    movel([0.104510, -1.367756, -2.579671, -0.764962, 1.570796, 1.675306],accel_mss,speed_ms,0,blend_radius_m)
    movel([0.104276, -1.367419, -2.579903, -0.765067, 1.570796, 1.675072],accel_mss,speed_ms,0,blend_radius_m)
    movel([0.103915, -1.367320, -2.579970, -0.765098, 1.570796, 1.674711],accel_mss,speed_ms,0,blend_radius_m)
    movel([0.103332, -1.367539, -2.579820, -0.765030, 1.570796, 1.674129],accel_mss,speed_ms,0,blend_radius_m)
    movel([0.102835, -1.367799, -2.579641, -0.764949, 1.570796, 1.673632],accel_mss,speed_ms,0,blend_radius_m)
    movel([0.102185, -1.368173, -2.579384, -0.764832, 1.570796, 1.672982],accel_mss,speed_ms,0,blend_radius_m)
    movel([0.099075, -1.369824, -2.578246, -0.764320, 1.570796, 1.669871],accel_mss,speed_ms,0,blend_radius_m)
    movel([0.095590, -1.371345, -2.577193, -0.763851, 1.570796, 1.666387],accel_mss,speed_ms,0,blend_radius_m)
    movel([0.091812, -1.372711, -2.576245, -0.763432, 1.570796, 1.662609],accel_mss,speed_ms,0,blend_radius_m)
    movel([0.087807, -1.373897, -2.575421, -0.763072, 1.570796, 1.658604],accel_mss,speed_ms,0,blend_radius_m)
    movel([0.084957, -1.374600, -2.574930, -0.762858, 1.570796, 1.655753],accel_mss,speed_ms,0,blend_radius_m)
    movel([0.082581, -1.375066, -2.574606, -0.762718, 1.570796, 1.653377],accel_mss,speed_ms,0,blend_radius_m)
    movel([0.080422, -1.375336, -2.574417, -0.762636, 1.570796, 1.651219],accel_mss,speed_ms,0,blend_radius_m)
    movel([0.078241, -1.375448, -2.574339, -0.762603, 1.570796, 1.649037],accel_mss,speed_ms,0,blend_radius_m)
    movel([0.077595, -1.375463, -2.574328, -0.762598, 1.570796, 1.648391],accel_mss,speed_ms,0,blend_radius_m)
    movel([0.077017, -1.375486, -2.574312, -0.762591, 1.570796, 1.647813],accel_mss,speed_ms,0,blend_radius_m)
    movel([0.076527, -1.375514, -2.574293, -0.762583, 1.570796, 1.647323],accel_mss,speed_ms,0,blend_radius_m)
    movel([0.076144, -1.375675, -2.574180, -0.762534, 1.570796, 1.646941],accel_mss,speed_ms,0,blend_radius_m)
    movel([0.075861, -1.375963, -2.573979, -0.762448, 1.570796, 1.646658],accel_mss,speed_ms,0,blend_radius_m)
    movel([0.075599, -1.376321, -2.573728, -0.762340, 1.570796, 1.646396],accel_mss,speed_ms,0,blend_radius_m)
    movel([0.075421, -1.376678, -2.573478, -0.762233, 1.570796, 1.646217],accel_mss,speed_ms,0,blend_radius_m)
    movel([0.075249, -1.377242, -2.573082, -0.762064, 1.570796, 1.646045],accel_mss,speed_ms,0,blend_radius_m)
    movel([0.075143, -1.377642, -2.572802, -0.761945, 1.570796, 1.645939],accel_mss,speed_ms,0,blend_radius_m)
    movel([0.075046, -1.378040, -2.572523, -0.761826, 1.570796, 1.645843],accel_mss,speed_ms,0,blend_radius_m)
    movel([0.074952, -1.378421, -2.572255, -0.761713, 1.570796, 1.645748],accel_mss,speed_ms,0,blend_radius_m)
    movel([0.074853, -1.378765, -2.572013, -0.761611, 1.570796, 1.645650],accel_mss,speed_ms,0,blend_radius_m)
    movel([0.074757, -1.379053, -2.571810, -0.761526, 1.570796, 1.645554],accel_mss,speed_ms,0,blend_radius_m)
    movel([0.074468, -1.379289, -2.571644, -0.761456, 1.570796, 1.645264],accel_mss,speed_ms,0,blend_radius_m)
    movel([0.073765, -1.379305, -2.571633, -0.761451, 1.570796, 1.644562],accel_mss,speed_ms,0,blend_radius_m)
    movel([0.073075, -1.379262, -2.571663, -0.761464, 1.570796, 1.643871],accel_mss,speed_ms,0,blend_radius_m)
    movel([0.072682, -1.379139, -2.571750, -0.761500, 1.570796, 1.643478],accel_mss,speed_ms,0,blend_radius_m)
    movel([0.072546, -1.379010, -2.571840, -0.761538, 1.570796, 1.643342],accel_mss,speed_ms,0,blend_radius_m)
    movel([0.072521, -1.378523, -2.572183, -0.761683, 1.570796, 1.643318],accel_mss,speed_ms,0,blend_radius_m)
    movel([0.072656, -1.377720, -2.572748, -0.761922, 1.570796, 1.643452],accel_mss,speed_ms,0,blend_radius_m)
    movel([0.073767, -1.373164, -2.575931, -0.763294, 1.570796, 1.644564],accel_mss,speed_ms,0,blend_radius_m)
    movel([0.075488, -1.368756, -2.578983, -0.764651, 1.570796, 1.646285],accel_mss,speed_ms,0,blend_radius_m)
    movel([0.077718, -1.364727, -2.581747, -0.765914, 1.570796, 1.648514],accel_mss,speed_ms,0,blend_radius_m)
    movel([0.080351, -1.361316, -2.584071, -0.767002, 1.570796, 1.651147],accel_mss,speed_ms,0,blend_radius_m)
    movel([0.082795, -1.358951, -2.585672, -0.767766, 1.570796, 1.653591],accel_mss,speed_ms,0,blend_radius_m)
    movel([0.085385, -1.357041, -2.586960, -0.768389, 1.570796, 1.656181],accel_mss,speed_ms,0,blend_radius_m)
    movel([0.088218, -1.355526, -2.587977, -0.768886, 1.570796, 1.659014],accel_mss,speed_ms,0,blend_radius_m)
    movel([0.091400, -1.354347, -2.588767, -0.769275, 1.570796, 1.662196],accel_mss,speed_ms,0,blend_radius_m)
    movel([0.094574, -1.353626, -2.589249, -0.769514, 1.570796, 1.665370],accel_mss,speed_ms,0,blend_radius_m)
    movel([0.097379, -1.353476, -2.589349, -0.769564, 1.570796, 1.668175],accel_mss,speed_ms,0,blend_radius_m)
    movel([0.099838, -1.353910, -2.589059, -0.769420, 1.570796, 1.670634],accel_mss,speed_ms,0,blend_radius_m)
    movel([0.101993, -1.354916, -2.588386, -0.769087, 1.570796, 1.672790],accel_mss,speed_ms,0,blend_radius_m)
    movel([0.103899, -1.356588, -2.587264, -0.768537, 1.570796, 1.674695],accel_mss,speed_ms,0,blend_radius_m)
    movel([0.105421, -1.358873, -2.585725, -0.767791, 1.570796, 1.676217],accel_mss,speed_ms,0,blend_radius_m)
    movel([0.106518, -1.361692, -2.583816, -0.766881, 1.570796, 1.677314],accel_mss,speed_ms,0,blend_radius_m)
    movel([0.107156, -1.364956, -2.581591, -0.765842, 1.570796, 1.677952],accel_mss,speed_ms,0,blend_radius_m)
    movel([0.107310, -1.366526, -2.580516, -0.765347, 1.570796, 1.678107],accel_mss,speed_ms,0,blend_radius_m)
    movel([0.107334, -1.367566, -2.579801, -0.765021, 1.570796, 1.678130],accel_mss,speed_ms,0,blend_radius_m)
    speed_ms = 0.003
    movel([0.107334, -1.370894, -2.581308, -0.760187, 1.570796, 1.678130],accel_mss,speed_ms,0,blend_radius_m)
    speed_ms = 0.007
    movel([0.107250, -1.371606, -2.580816, -0.759967, 1.570796, 1.678047],accel_mss,speed_ms,0,blend_radius_m)
    movel([0.107024, -1.371990, -2.580550, -0.759849, 1.570796, 1.677820],accel_mss,speed_ms,0,blend_radius_m)
    movel([0.106591, -1.372345, -2.580304, -0.759740, 1.570796, 1.677388],accel_mss,speed_ms,0,blend_radius_m)
    movel([0.105893, -1.372818, -2.579976, -0.759595, 1.570796, 1.676689],accel_mss,speed_ms,0,blend_radius_m)
    movel([0.105181, -1.373264, -2.579667, -0.759459, 1.570796, 1.675977],accel_mss,speed_ms,0,blend_radius_m)
    movel([0.104870, -1.373304, -2.579639, -0.759446, 1.570796, 1.675666],accel_mss,speed_ms,0,blend_radius_m)
    movel([0.104761, -1.373118, -2.579768, -0.759503, 1.570796, 1.675557],accel_mss,speed_ms,0,blend_radius_m)
    movel([0.104653, -1.371747, -2.580718, -0.759924, 1.570796, 1.675449],accel_mss,speed_ms,0,blend_radius_m)
    movel([0.104510, -1.371083, -2.581178, -0.760128, 1.570796, 1.675306],accel_mss,speed_ms,0,blend_radius_m)
    movel([0.104276, -1.370747, -2.581410, -0.760232, 1.570796, 1.675072],accel_mss,speed_ms,0,blend_radius_m)
    movel([0.103915, -1.370648, -2.581478, -0.760263, 1.570796, 1.674711],accel_mss,speed_ms,0,blend_radius_m)
    movel([0.103332, -1.370866, -2.581327, -0.760195, 1.570796, 1.674129],accel_mss,speed_ms,0,blend_radius_m)
    movel([0.102835, -1.371126, -2.581148, -0.760115, 1.570796, 1.673632],accel_mss,speed_ms,0,blend_radius_m)
    movel([0.102185, -1.371499, -2.580890, -0.760000, 1.570796, 1.672982],accel_mss,speed_ms,0,blend_radius_m)
    movel([0.099075, -1.373145, -2.579749, -0.759495, 1.570796, 1.669871],accel_mss,speed_ms,0,blend_radius_m)
    movel([0.095590, -1.374663, -2.578694, -0.759032, 1.570796, 1.666387],accel_mss,speed_ms,0,blend_radius_m)
    movel([0.091812, -1.376025, -2.577744, -0.758620, 1.570796, 1.662609],accel_mss,speed_ms,0,blend_radius_m)
    movel([0.087807, -1.377207, -2.576917, -0.758264, 1.570796, 1.658604],accel_mss,speed_ms,0,blend_radius_m)
    movel([0.084957, -1.377909, -2.576426, -0.758054, 1.570796, 1.655753],accel_mss,speed_ms,0,blend_radius_m)
    movel([0.082581, -1.378373, -2.576100, -0.757916, 1.570796, 1.653377],accel_mss,speed_ms,0,blend_radius_m)
    movel([0.080422, -1.378642, -2.575911, -0.757835, 1.570796, 1.651219],accel_mss,speed_ms,0,blend_radius_m)
    movel([0.078241, -1.378754, -2.575833, -0.757802, 1.570796, 1.649037],accel_mss,speed_ms,0,blend_radius_m)
    movel([0.077595, -1.378769, -2.575822, -0.757798, 1.570796, 1.648391],accel_mss,speed_ms,0,blend_radius_m)
    movel([0.077017, -1.378792, -2.575806, -0.757791, 1.570796, 1.647813],accel_mss,speed_ms,0,blend_radius_m)
    movel([0.076527, -1.378820, -2.575787, -0.757783, 1.570796, 1.647323],accel_mss,speed_ms,0,blend_radius_m)
    movel([0.076144, -1.378981, -2.575673, -0.757735, 1.570796, 1.646941],accel_mss,speed_ms,0,blend_radius_m)
    movel([0.075861, -1.379268, -2.575472, -0.757649, 1.570796, 1.646658],accel_mss,speed_ms,0,blend_radius_m)
    movel([0.075599, -1.379625, -2.575220, -0.757543, 1.570796, 1.646396],accel_mss,speed_ms,0,blend_radius_m)
    movel([0.075421, -1.379981, -2.574970, -0.757438, 1.570796, 1.646217],accel_mss,speed_ms,0,blend_radius_m)
    movel([0.075249, -1.380544, -2.574573, -0.757272, 1.570796, 1.646045],accel_mss,speed_ms,0,blend_radius_m)
    movel([0.075143, -1.380942, -2.574293, -0.757154, 1.570796, 1.645939],accel_mss,speed_ms,0,blend_radius_m)
    movel([0.075046, -1.381339, -2.574012, -0.757037, 1.570796, 1.645843],accel_mss,speed_ms,0,blend_radius_m)
    movel([0.074952, -1.381719, -2.573744, -0.756926, 1.570796, 1.645748],accel_mss,speed_ms,0,blend_radius_m)
    movel([0.074853, -1.382062, -2.573502, -0.756825, 1.570796, 1.645650],accel_mss,speed_ms,0,blend_radius_m)
    movel([0.074757, -1.382350, -2.573298, -0.756741, 1.570796, 1.645554],accel_mss,speed_ms,0,blend_radius_m)
    movel([0.074468, -1.382585, -2.573132, -0.756672, 1.570796, 1.645264],accel_mss,speed_ms,0,blend_radius_m)
    movel([0.073765, -1.382601, -2.573121, -0.756668, 1.570796, 1.644562],accel_mss,speed_ms,0,blend_radius_m)
    movel([0.073075, -1.382558, -2.573151, -0.756680, 1.570796, 1.643871],accel_mss,speed_ms,0,blend_radius_m)
    movel([0.072682, -1.382435, -2.573238, -0.756716, 1.570796, 1.643478],accel_mss,speed_ms,0,blend_radius_m)
    movel([0.072546, -1.382307, -2.573329, -0.756753, 1.570796, 1.643342],accel_mss,speed_ms,0,blend_radius_m)
    movel([0.072521, -1.381821, -2.573672, -0.756896, 1.570796, 1.643318],accel_mss,speed_ms,0,blend_radius_m)
    movel([0.072656, -1.381020, -2.574238, -0.757131, 1.570796, 1.643452],accel_mss,speed_ms,0,blend_radius_m)
    movel([0.073767, -1.376476, -2.577429, -0.758484, 1.570796, 1.644564],accel_mss,speed_ms,0,blend_radius_m)
    movel([0.075488, -1.372080, -2.580488, -0.759821, 1.570796, 1.646285],accel_mss,speed_ms,0,blend_radius_m)
    movel([0.077718, -1.368062, -2.583259, -0.761067, 1.570796, 1.648514],accel_mss,speed_ms,0,blend_radius_m)
    movel([0.080351, -1.364660, -2.585588, -0.762141, 1.570796, 1.651147],accel_mss,speed_ms,0,blend_radius_m)
    movel([0.082795, -1.362302, -2.587193, -0.762894, 1.570796, 1.653591],accel_mss,speed_ms,0,blend_radius_m)
    movel([0.085385, -1.360396, -2.588484, -0.763509, 1.570796, 1.656181],accel_mss,speed_ms,0,blend_radius_m)
    movel([0.088218, -1.358885, -2.589504, -0.764000, 1.570796, 1.659014],accel_mss,speed_ms,0,blend_radius_m)
    movel([0.091400, -1.357709, -2.590296, -0.764384, 1.570796, 1.662196],accel_mss,speed_ms,0,blend_radius_m)
    movel([0.094574, -1.356990, -2.590779, -0.764620, 1.570796, 1.665370],accel_mss,speed_ms,0,blend_radius_m)
    movel([0.097379, -1.356841, -2.590879, -0.764669, 1.570796, 1.668175],accel_mss,speed_ms,0,blend_radius_m)
    movel([0.099838, -1.357273, -2.590589, -0.764527, 1.570796, 1.670634],accel_mss,speed_ms,0,blend_radius_m)
    movel([0.101993, -1.358277, -2.589914, -0.764198, 1.570796, 1.672790],accel_mss,speed_ms,0,blend_radius_m)
    movel([0.103899, -1.359945, -2.588789, -0.763655, 1.570796, 1.674695],accel_mss,speed_ms,0,blend_radius_m)
    movel([0.105421, -1.362224, -2.587246, -0.762919, 1.570796, 1.676217],accel_mss,speed_ms,0,blend_radius_m)
    movel([0.106518, -1.365035, -2.585333, -0.762022, 1.570796, 1.677314],accel_mss,speed_ms,0,blend_radius_m)
    movel([0.107156, -1.368290, -2.583103, -0.760996, 1.570796, 1.677952],accel_mss,speed_ms,0,blend_radius_m)
    movel([0.107310, -1.369856, -2.582025, -0.760508, 1.570796, 1.678107],accel_mss,speed_ms,0,blend_radius_m)
    movel([0.107334, -1.370894, -2.581308, -0.760187, 1.570796, 1.678130],accel_mss,speed_ms,0,blend_radius_m)
    speed_ms = 0.003
    movel([0.107334, -1.357724, -2.575230, -0.779436, 1.570796, 1.678130],accel_mss,speed_ms,0,blend_radius_m)
    speed_ms = 1.000
    movel([0.107334, -1.332493, -2.562679, -0.817217, 1.570796, 1.678130],accel_mss,speed_ms,0,blend_radius_m)
    movel([0.108777, -1.323962, -2.568202, -0.820226, 1.570796, 1.679573],accel_mss,speed_ms,0,blend_radius_m)
    movel([0.108777, -1.349338, -2.580862, -0.782189, 1.570796, 1.679573],accel_mss,speed_ms,0,blend_radius_m)
    speed_ms = 0.003
    movel([0.108777, -1.359243, -2.585475, -0.767671, 1.570796, 1.679573],accel_mss,speed_ms,0,blend_radius_m)
    speed_ms = 0.007
    speed_ms = 0.003
    movel([0.108777, -1.362592, -2.586996, -0.762801, 1.570796, 1.679573],accel_mss,speed_ms,0,blend_radius_m)
    speed_ms = 0.007
    speed_ms = 0.003
    movel([0.108777, -1.349338, -2.580862, -0.782189, 1.570796, 1.679573],accel_mss,speed_ms,0,blend_radius_m)
    speed_ms = 1.000
    movel([0.108777, -1.323962, -2.568202, -0.820226, 1.570796, 1.679573],accel_mss,speed_ms,0,blend_radius_m)
    movel([0.115883, -1.313834, -2.574634, -0.823920, 1.570796, 1.686679],accel_mss,speed_ms,0,blend_radius_m)
    movel([0.115883, -1.339378, -2.587426, -0.785585, 1.570796, 1.686679],accel_mss,speed_ms,0,blend_radius_m)
    speed_ms = 0.003
    movel([0.115883, -1.349357, -2.592088, -0.770944, 1.570796, 1.686679],accel_mss,speed_ms,0,blend_radius_m)
    speed_ms = 0.007
    movel([0.115699, -1.349014, -2.592315, -0.771060, 1.570796, 1.686495],accel_mss,speed_ms,0,blend_radius_m)
    movel([0.115676, -1.348698, -2.592524, -0.771167, 1.570796, 1.686472],accel_mss,speed_ms,0,blend_radius_m)
    movel([0.115575, -1.348533, -2.592633, -0.771223, 1.570796, 1.686372],accel_mss,speed_ms,0,blend_radius_m)
    movel([0.115017, -1.348527, -2.592637, -0.771225, 1.570796, 1.685813],accel_mss,speed_ms,0,blend_radius_m)
    movel([0.114668, -1.348560, -2.592615, -0.771214, 1.570796, 1.685464],accel_mss,speed_ms,0,blend_radius_m)
    movel([0.114704, -1.348286, -2.592796, -0.771307, 1.570796, 1.685500],accel_mss,speed_ms,0,blend_radius_m)
    movel([0.115071, -1.348116, -2.592908, -0.771365, 1.570796, 1.685867],accel_mss,speed_ms,0,blend_radius_m)
    movel([0.115442, -1.347956, -2.593014, -0.771419, 1.570796, 1.686238],accel_mss,speed_ms,0,blend_radius_m)
    movel([0.115828, -1.347543, -2.593286, -0.771560, 1.570796, 1.686625],accel_mss,speed_ms,0,blend_radius_m)
    movel([0.115940, -1.347188, -2.593520, -0.771680, 1.570796, 1.686737],accel_mss,speed_ms,0,blend_radius_m)
    movel([0.116063, -1.346865, -2.593733, -0.771791, 1.570796, 1.686859],accel_mss,speed_ms,0,blend_radius_m)
    movel([0.116375, -1.346777, -2.593791, -0.771821, 1.570796, 1.687171],accel_mss,speed_ms,0,blend_radius_m)
    movel([0.116418, -1.347053, -2.593609, -0.771727, 1.570796, 1.687215],accel_mss,speed_ms,0,blend_radius_m)
    movel([0.116441, -1.347370, -2.593400, -0.771619, 1.570796, 1.687238],accel_mss,speed_ms,0,blend_radius_m)
    movel([0.116544, -1.347537, -2.593291, -0.771562, 1.570796, 1.687340],accel_mss,speed_ms,0,blend_radius_m)
    movel([0.117057, -1.347533, -2.593293, -0.771563, 1.570796, 1.687853],accel_mss,speed_ms,0,blend_radius_m)
    movel([0.117373, -1.347465, -2.593337, -0.771586, 1.570796, 1.688169],accel_mss,speed_ms,0,blend_radius_m)
    movel([0.117594, -1.347568, -2.593270, -0.771551, 1.570796, 1.688390],accel_mss,speed_ms,0,blend_radius_m)
    movel([0.117342, -1.347828, -2.593098, -0.771463, 1.570796, 1.688138],accel_mss,speed_ms,0,blend_radius_m)
    movel([0.117058, -1.347954, -2.593015, -0.771420, 1.570796, 1.687854],accel_mss,speed_ms,0,blend_radius_m)
    movel([0.116674, -1.348120, -2.592906, -0.771363, 1.570796, 1.687470],accel_mss,speed_ms,0,blend_radius_m)
    movel([0.116280, -1.348525, -2.592638, -0.771226, 1.570796, 1.687077],accel_mss,speed_ms,0,blend_radius_m)
    movel([0.116173, -1.348860, -2.592416, -0.771112, 1.570796, 1.686970],accel_mss,speed_ms,0,blend_radius_m)
    movel([0.116055, -1.349207, -2.592187, -0.770995, 1.570796, 1.686851],accel_mss,speed_ms,0,blend_radius_m)
    speed_ms = 0.003
    movel([0.115883, -1.352732, -2.593625, -0.766032, 1.570796, 1.686679],accel_mss,speed_ms,0,blend_radius_m)
    speed_ms = 0.007
    movel([0.115699, -1.352390, -2.593853, -0.766147, 1.570796, 1.686495],accel_mss,speed_ms,0,blend_radius_m)
    movel([0.115676, -1.352075, -2.594062, -0.766252, 1.570796, 1.686472],accel_mss,speed_ms,0,blend_radius_m)
    movel([0.115575, -1.351910, -2.594171, -0.766307, 1.570796, 1.686372],accel_mss,speed_ms,0,blend_radius_m)
    movel([0.115017, -1.351904, -2.594176, -0.766310, 1.570796, 1.685813],accel_mss,speed_ms,0,blend_radius_m)
    movel([0.114668, -1.351937, -2.594154, -0.766299, 1.570796, 1.685464],accel_mss,speed_ms,0,blend_radius_m)
    movel([0.114704, -1.351664, -2.594335, -0.766390, 1.570796, 1.685500],accel_mss,speed_ms,0,blend_radius_m)
    movel([0.115071, -1.351494, -2.594447, -0.766447, 1.570796, 1.685867],accel_mss,speed_ms,0,blend_radius_m)
    movel([0.115442, -1.351335, -2.594553, -0.766501, 1.570796, 1.686238],accel_mss,speed_ms,0,blend_radius_m)
    movel([0.115828, -1.350923, -2.594826, -0.766640, 1.570796, 1.686625],accel_mss,speed_ms,0,blend_radius_m)
    movel([0.115940, -1.350569, -2.595061, -0.766759, 1.570796, 1.686737],accel_mss,speed_ms,0,blend_radius_m)
    movel([0.116063, -1.350247, -2.595274, -0.766868, 1.570796, 1.686859],accel_mss,speed_ms,0,blend_radius_m)
    movel([0.116375, -1.350159, -2.595333, -0.766898, 1.570796, 1.687171],accel_mss,speed_ms,0,blend_radius_m)
    movel([0.116418, -1.350434, -2.595150, -0.766805, 1.570796, 1.687215],accel_mss,speed_ms,0,blend_radius_m)
    movel([0.116441, -1.350750, -2.594941, -0.766698, 1.570796, 1.687238],accel_mss,speed_ms,0,blend_radius_m)
    movel([0.116544, -1.350916, -2.594831, -0.766642, 1.570796, 1.687340],accel_mss,speed_ms,0,blend_radius_m)
    movel([0.117057, -1.350912, -2.594833, -0.766643, 1.570796, 1.687853],accel_mss,speed_ms,0,blend_radius_m)
    movel([0.117373, -1.350845, -2.594878, -0.766666, 1.570796, 1.688169],accel_mss,speed_ms,0,blend_radius_m)
    movel([0.117594, -1.350948, -2.594810, -0.766631, 1.570796, 1.688390],accel_mss,speed_ms,0,blend_radius_m)
    movel([0.117342, -1.351207, -2.594638, -0.766544, 1.570796, 1.688138],accel_mss,speed_ms,0,blend_radius_m)
    movel([0.117058, -1.351333, -2.594555, -0.766501, 1.570796, 1.687854],accel_mss,speed_ms,0,blend_radius_m)
    movel([0.116674, -1.351498, -2.594445, -0.766446, 1.570796, 1.687470],accel_mss,speed_ms,0,blend_radius_m)
    movel([0.116280, -1.351902, -2.594177, -0.766310, 1.570796, 1.687077],accel_mss,speed_ms,0,blend_radius_m)
    movel([0.116173, -1.352237, -2.593954, -0.766198, 1.570796, 1.686970],accel_mss,speed_ms,0,blend_radius_m)
    movel([0.116055, -1.352583, -2.593724, -0.766082, 1.570796, 1.686851],accel_mss,speed_ms,0,blend_radius_m)
    speed_ms = 0.003
    movel([0.115883, -1.339378, -2.587426, -0.785585, 1.570796, 1.686679],accel_mss,speed_ms,0,blend_radius_m)
    speed_ms = 1.000
    movel([0.115883, -1.313834, -2.574634, -0.823920, 1.570796, 1.686679],accel_mss,speed_ms,0,blend_radius_m)
    movel([0.116165, -1.307823, -2.578390, -0.826176, 1.570796, 1.686961],accel_mss,speed_ms,0,blend_radius_m)
    movel([0.116165, -1.333465, -2.591259, -0.787665, 1.570796, 1.686961],accel_mss,speed_ms,0,blend_radius_m)
    speed_ms = 0.003
    movel([0.116165, -1.343486, -2.595951, -0.772952, 1.570796, 1.686961],accel_mss,speed_ms,0,blend_radius_m)
    speed_ms = 0.007
    movel([0.115451, -1.343685, -2.595821, -0.772883, 1.570796, 1.686247],accel_mss,speed_ms,0,blend_radius_m)
    movel([0.115104, -1.343689, -2.595818, -0.772882, 1.570796, 1.685900],accel_mss,speed_ms,0,blend_radius_m)
    movel([0.115268, -1.343302, -2.596071, -0.773016, 1.570796, 1.686064],accel_mss,speed_ms,0,blend_radius_m)
    movel([0.115501, -1.343098, -2.596204, -0.773087, 1.570796, 1.686297],accel_mss,speed_ms,0,blend_radius_m)
    movel([0.115888, -1.342901, -2.596333, -0.773155, 1.570796, 1.686685],accel_mss,speed_ms,0,blend_radius_m)
    movel([0.116623, -1.342625, -2.596513, -0.773251, 1.570796, 1.687420],accel_mss,speed_ms,0,blend_radius_m)
    movel([0.117131, -1.342452, -2.596626, -0.773311, 1.570796, 1.687928],accel_mss,speed_ms,0,blend_radius_m)
    movel([0.117489, -1.342352, -2.596691, -0.773346, 1.570796, 1.688285],accel_mss,speed_ms,0,blend_radius_m)
    movel([0.117872, -1.342327, -2.596707, -0.773354, 1.570796, 1.688668],accel_mss,speed_ms,0,blend_radius_m)
    movel([0.118205, -1.342164, -2.596814, -0.773411, 1.570796, 1.689001],accel_mss,speed_ms,0,blend_radius_m)
    movel([0.118288, -1.342353, -2.596691, -0.773345, 1.570796, 1.689084],accel_mss,speed_ms,0,blend_radius_m)
    movel([0.117936, -1.342765, -2.596422, -0.773202, 1.570796, 1.688732],accel_mss,speed_ms,0,blend_radius_m)
    movel([0.117499, -1.343009, -2.596262, -0.773117, 1.570796, 1.688295],accel_mss,speed_ms,0,blend_radius_m)
    movel([0.116912, -1.343249, -2.596106, -0.773034, 1.570796, 1.687708],accel_mss,speed_ms,0,blend_radius_m)
    movel([0.116165, -1.343486, -2.595951, -0.772952, 1.570796, 1.686961],accel_mss,speed_ms,0,blend_radius_m)
    speed_ms = 0.003
    movel([0.116165, -1.346876, -2.597498, -0.768015, 1.570796, 1.686961],accel_mss,speed_ms,0,blend_radius_m)
    speed_ms = 0.007
    movel([0.115451, -1.347074, -2.597367, -0.767947, 1.570796, 1.686247],accel_mss,speed_ms,0,blend_radius_m)
    movel([0.115104, -1.347078, -2.597365, -0.767946, 1.570796, 1.685900],accel_mss,speed_ms,0,blend_radius_m)
    movel([0.115268, -1.346692, -2.597619, -0.768078, 1.570796, 1.686064],accel_mss,speed_ms,0,blend_radius_m)
    movel([0.115501, -1.346489, -2.597752, -0.768148, 1.570796, 1.686297],accel_mss,speed_ms,0,blend_radius_m)
    movel([0.115888, -1.346292, -2.597881, -0.768215, 1.570796, 1.686685],accel_mss,speed_ms,0,blend_radius_m)
    movel([0.116623, -1.346017, -2.598062, -0.768310, 1.570796, 1.687420],accel_mss,speed_ms,0,blend_radius_m)
    movel([0.117131, -1.345844, -2.598175, -0.768370, 1.570796, 1.687928],accel_mss,speed_ms,0,blend_radius_m)
    movel([0.117489, -1.345745, -2.598240, -0.768404, 1.570796, 1.688285],accel_mss,speed_ms,0,blend_radius_m)
    movel([0.117872, -1.345720, -2.598256, -0.768412, 1.570796, 1.688668],accel_mss,speed_ms,0,blend_radius_m)
    movel([0.118205, -1.345557, -2.598363, -0.768468, 1.570796, 1.689001],accel_mss,speed_ms,0,blend_radius_m)
    movel([0.118288, -1.345746, -2.598240, -0.768403, 1.570796, 1.689084],accel_mss,speed_ms,0,blend_radius_m)
    movel([0.117936, -1.346157, -2.597970, -0.768262, 1.570796, 1.688732],accel_mss,speed_ms,0,blend_radius_m)
    movel([0.117499, -1.346400, -2.597810, -0.768178, 1.570796, 1.688295],accel_mss,speed_ms,0,blend_radius_m)
    movel([0.116912, -1.346639, -2.597653, -0.768096, 1.570796, 1.687708],accel_mss,speed_ms,0,blend_radius_m)
    movel([0.116165, -1.346876, -2.597498, -0.768015, 1.570796, 1.686961],accel_mss,speed_ms,0,blend_radius_m)
    speed_ms = 0.003
    movel([0.116165, -1.333465, -2.591259, -0.787665, 1.570796, 1.686961],accel_mss,speed_ms,0,blend_radius_m)
    speed_ms = 1.000
    movel([0.116165, -1.307823, -2.578390, -0.826176, 1.570796, 1.686961],accel_mss,speed_ms,0,blend_radius_m)
    movel([0.116275, -1.306704, -2.579085, -0.826601, 1.570796, 1.687071],accel_mss,speed_ms,0,blend_radius_m)
    movel([0.116275, -1.332363, -2.591968, -0.788057, 1.570796, 1.687071],accel_mss,speed_ms,0,blend_radius_m)
    speed_ms = 0.003
    movel([0.116275, -1.342392, -2.596665, -0.773332, 1.570796, 1.687071],accel_mss,speed_ms,0,blend_radius_m)
    speed_ms = 0.007
    movel([0.114992, -1.342821, -2.596385, -0.773183, 1.570796, 1.685788],accel_mss,speed_ms,0,blend_radius_m)
    movel([0.115029, -1.342536, -2.596571, -0.773282, 1.570796, 1.685826],accel_mss,speed_ms,0,blend_radius_m)
    movel([0.115135, -1.342289, -2.596733, -0.773368, 1.570796, 1.685931],accel_mss,speed_ms,0,blend_radius_m)
    movel([0.115455, -1.341882, -2.596998, -0.773509, 1.570796, 1.686251],accel_mss,speed_ms,0,blend_radius_m)
    movel([0.115812, -1.341501, -2.597246, -0.773642, 1.570796, 1.686608],accel_mss,speed_ms,0,blend_radius_m)
    movel([0.116087, -1.341342, -2.597350, -0.773697, 1.570796, 1.686883],accel_mss,speed_ms,0,blend_radius_m)
    movel([0.116501, -1.341104, -2.597505, -0.773780, 1.570796, 1.687297],accel_mss,speed_ms,0,blend_radius_m)
    movel([0.117092, -1.340955, -2.597601, -0.773833, 1.570796, 1.687889],accel_mss,speed_ms,0,blend_radius_m)
    movel([0.117675, -1.340833, -2.597681, -0.773875, 1.570796, 1.688471],accel_mss,speed_ms,0,blend_radius_m)
    movel([0.117918, -1.340842, -2.597675, -0.773872, 1.570796, 1.688714],accel_mss,speed_ms,0,blend_radius_m)
    movel([0.118172, -1.340876, -2.597653, -0.773860, 1.570796, 1.688969],accel_mss,speed_ms,0,blend_radius_m)
    movel([0.118369, -1.340949, -2.597606, -0.773835, 1.570796, 1.689165],accel_mss,speed_ms,0,blend_radius_m)
    movel([0.118272, -1.341334, -2.597355, -0.773700, 1.570796, 1.689068],accel_mss,speed_ms,0,blend_radius_m)
    movel([0.118052, -1.341618, -2.597170, -0.773601, 1.570796, 1.688849],accel_mss,speed_ms,0,blend_radius_m)
    movel([0.117694, -1.341850, -2.597018, -0.773520, 1.570796, 1.688491],accel_mss,speed_ms,0,blend_radius_m)
    movel([0.117282, -1.342023, -2.596906, -0.773460, 1.570796, 1.688078],accel_mss,speed_ms,0,blend_radius_m)
    movel([0.116789, -1.342212, -2.596782, -0.773394, 1.570796, 1.687585],accel_mss,speed_ms,0,blend_radius_m)
    movel([0.116275, -1.342392, -2.596665, -0.773332, 1.570796, 1.687071],accel_mss,speed_ms,0,blend_radius_m)
    speed_ms = 0.003
    movel([0.116275, -1.345785, -2.598214, -0.768390, 1.570796, 1.687071],accel_mss,speed_ms,0,blend_radius_m)
    speed_ms = 0.007
    movel([0.114992, -1.346213, -2.597934, -0.768243, 1.570796, 1.685788],accel_mss,speed_ms,0,blend_radius_m)
    movel([0.115029, -1.345928, -2.598120, -0.768341, 1.570796, 1.685826],accel_mss,speed_ms,0,blend_radius_m)
    movel([0.115135, -1.345682, -2.598282, -0.768426, 1.570796, 1.685931],accel_mss,speed_ms,0,blend_radius_m)
    movel([0.115455, -1.345276, -2.598547, -0.768565, 1.570796, 1.686251],accel_mss,speed_ms,0,blend_radius_m)
    movel([0.115812, -1.344896, -2.598797, -0.768697, 1.570796, 1.686608],accel_mss,speed_ms,0,blend_radius_m)
    movel([0.116087, -1.344738, -2.598900, -0.768751, 1.570796, 1.686883],accel_mss,speed_ms,0,blend_radius_m)
    movel([0.116501, -1.344500, -2.599056, -0.768833, 1.570796, 1.687297],accel_mss,speed_ms,0,blend_radius_m)
    movel([0.117092, -1.344351, -2.599153, -0.768885, 1.570796, 1.687889],accel_mss,speed_ms,0,blend_radius_m)
    movel([0.117675, -1.344230, -2.599232, -0.768927, 1.570796, 1.688471],accel_mss,speed_ms,0,blend_radius_m)
    movel([0.117918, -1.344238, -2.599227, -0.768924, 1.570796, 1.688714],accel_mss,speed_ms,0,blend_radius_m)
    movel([0.118172, -1.344272, -2.599204, -0.768912, 1.570796, 1.688969],accel_mss,speed_ms,0,blend_radius_m)
    movel([0.118369, -1.344345, -2.599157, -0.768887, 1.570796, 1.689165],accel_mss,speed_ms,0,blend_radius_m)
    movel([0.118272, -1.344729, -2.598906, -0.768754, 1.570796, 1.689068],accel_mss,speed_ms,0,blend_radius_m)
    movel([0.118052, -1.345012, -2.598720, -0.768656, 1.570796, 1.688849],accel_mss,speed_ms,0,blend_radius_m)
    movel([0.117694, -1.345244, -2.598568, -0.768576, 1.570796, 1.688491],accel_mss,speed_ms,0,blend_radius_m)
    movel([0.117282, -1.345417, -2.598455, -0.768517, 1.570796, 1.688078],accel_mss,speed_ms,0,blend_radius_m)
    movel([0.116789, -1.345606, -2.598332, -0.768452, 1.570796, 1.687585],accel_mss,speed_ms,0,blend_radius_m)
    movel([0.116275, -1.345785, -2.598214, -0.768390, 1.570796, 1.687071],accel_mss,speed_ms,0,blend_radius_m)
    speed_ms = 0.003
    movel([0.116275, -1.332363, -2.591968, -0.788057, 1.570796, 1.687071],accel_mss,speed_ms,0,blend_radius_m)
    speed_ms = 1.000
    movel([0.116275, -1.306704, -2.579085, -0.826601, 1.570796, 1.687071],accel_mss,speed_ms,0,blend_radius_m)
    movel([0.110311, -1.309407, -2.577405, -0.825577, 1.570796, 1.681108],accel_mss,speed_ms,0,blend_radius_m)
    movel([0.110311, -1.335023, -2.590253, -0.787112, 1.570796, 1.681108],accel_mss,speed_ms,0,blend_radius_m)
    speed_ms = 0.003
    movel([0.110311, -1.345033, -2.594937, -0.772418, 1.570796, 1.681108],accel_mss,speed_ms,0,blend_radius_m)
    speed_ms = 0.007
    movel([0.110218, -1.345333, -2.594740, -0.772315, 1.570796, 1.681015],accel_mss,speed_ms,0,blend_radius_m)
    movel([0.110038, -1.345690, -2.594506, -0.772193, 1.570796, 1.680834],accel_mss,speed_ms,0,blend_radius_m)
    movel([0.109560, -1.346240, -2.594145, -0.772005, 1.570796, 1.680356],accel_mss,speed_ms,0,blend_radius_m)
    movel([0.108920, -1.346642, -2.593880, -0.771867, 1.570796, 1.679717],accel_mss,speed_ms,0,blend_radius_m)
    movel([0.108265, -1.346808, -2.593771, -0.771810, 1.570796, 1.679062],accel_mss,speed_ms,0,blend_radius_m)
    movel([0.107740, -1.346699, -2.593843, -0.771848, 1.570796, 1.678536],accel_mss,speed_ms,0,blend_radius_m)
    movel([0.107409, -1.346368, -2.594060, -0.771961, 1.570796, 1.678205],accel_mss,speed_ms,0,blend_radius_m)
    movel([0.107327, -1.345934, -2.594346, -0.772109, 1.570796, 1.678123],accel_mss,speed_ms,0,blend_radius_m)
    movel([0.107509, -1.345417, -2.594686, -0.772287, 1.570796, 1.678305],accel_mss,speed_ms,0,blend_radius_m)
    movel([0.107937, -1.344853, -2.595055, -0.772480, 1.570796, 1.678734],accel_mss,speed_ms,0,blend_radius_m)
    movel([0.108340, -1.344485, -2.595297, -0.772607, 1.570796, 1.679136],accel_mss,speed_ms,0,blend_radius_m)
    movel([0.108727, -1.344242, -2.595456, -0.772691, 1.570796, 1.679523],accel_mss,speed_ms,0,blend_radius_m)
    movel([0.109109, -1.344122, -2.595535, -0.772732, 1.570796, 1.679905],accel_mss,speed_ms,0,blend_radius_m)
    movel([0.109499, -1.344117, -2.595538, -0.772734, 1.570796, 1.680296],accel_mss,speed_ms,0,blend_radius_m)
    movel([0.109823, -1.344224, -2.595468, -0.772697, 1.570796, 1.680619],accel_mss,speed_ms,0,blend_radius_m)
    movel([0.110099, -1.344446, -2.595322, -0.772621, 1.570796, 1.680895],accel_mss,speed_ms,0,blend_radius_m)
    movel([0.110276, -1.344735, -2.595133, -0.772521, 1.570796, 1.681072],accel_mss,speed_ms,0,blend_radius_m)
    movel([0.110311, -1.345033, -2.594937, -0.772418, 1.570796, 1.681108],accel_mss,speed_ms,0,blend_radius_m)
    speed_ms = 0.003
    movel([0.110311, -1.348419, -2.596482, -0.767488, 1.570796, 1.681108],accel_mss,speed_ms,0,blend_radius_m)
    speed_ms = 0.007
    movel([0.110218, -1.348719, -2.596284, -0.767386, 1.570796, 1.681015],accel_mss,speed_ms,0,blend_radius_m)
    movel([0.110038, -1.349074, -2.596050, -0.767265, 1.570796, 1.680834],accel_mss,speed_ms,0,blend_radius_m)
    movel([0.109560, -1.349623, -2.595687, -0.767079, 1.570796, 1.680356],accel_mss,speed_ms,0,blend_radius_m)
    movel([0.108920, -1.350024, -2.595422, -0.766943, 1.570796, 1.679717],accel_mss,speed_ms,0,blend_radius_m)
    movel([0.108265, -1.350189, -2.595312, -0.766887, 1.570796, 1.679062],accel_mss,speed_ms,0,blend_radius_m)
    movel([0.107740, -1.350080, -2.595384, -0.766924, 1.570796, 1.678536],accel_mss,speed_ms,0,blend_radius_m)
    movel([0.107409, -1.349751, -2.595603, -0.767036, 1.570796, 1.678205],accel_mss,speed_ms,0,blend_radius_m)
    movel([0.107327, -1.349318, -2.595889, -0.767182, 1.570796, 1.678123],accel_mss,speed_ms,0,blend_radius_m)
    movel([0.107509, -1.348802, -2.596229, -0.767358, 1.570796, 1.678305],accel_mss,speed_ms,0,blend_radius_m)
    movel([0.107937, -1.348240, -2.596600, -0.767549, 1.570796, 1.678734],accel_mss,speed_ms,0,blend_radius_m)
    movel([0.108340, -1.347872, -2.596842, -0.767675, 1.570796, 1.679136],accel_mss,speed_ms,0,blend_radius_m)
    movel([0.108727, -1.347630, -2.597002, -0.767757, 1.570796, 1.679523],accel_mss,speed_ms,0,blend_radius_m)
    movel([0.109109, -1.347510, -2.597081, -0.767798, 1.570796, 1.679905],accel_mss,speed_ms,0,blend_radius_m)
    movel([0.109499, -1.347505, -2.597084, -0.767800, 1.570796, 1.680296],accel_mss,speed_ms,0,blend_radius_m)
    movel([0.109823, -1.347612, -2.597014, -0.767763, 1.570796, 1.680619],accel_mss,speed_ms,0,blend_radius_m)
    movel([0.110099, -1.347834, -2.596868, -0.767688, 1.570796, 1.680895],accel_mss,speed_ms,0,blend_radius_m)
    movel([0.110276, -1.348121, -2.596678, -0.767589, 1.570796, 1.681072],accel_mss,speed_ms,0,blend_radius_m)
    movel([0.110311, -1.348419, -2.596482, -0.767488, 1.570796, 1.681108],accel_mss,speed_ms,0,blend_radius_m)
    speed_ms = 0.003
    movel([0.110311, -1.335023, -2.590253, -0.787112, 1.570796, 1.681108],accel_mss,speed_ms,0,blend_radius_m)
    speed_ms = 1.000
    movel([0.110311, -1.309407, -2.577405, -0.825577, 1.570796, 1.681108],accel_mss,speed_ms,0,blend_radius_m)
    movel([0.104721, -1.314744, -2.574062, -0.823583, 1.570796, 1.675517],accel_mss,speed_ms,0,blend_radius_m)
    movel([0.104721, -1.340273, -2.586841, -0.785274, 1.570796, 1.675517],accel_mss,speed_ms,0,blend_radius_m)
    speed_ms = 0.003
    movel([0.104721, -1.350245, -2.591499, -0.770645, 1.570796, 1.675517],accel_mss,speed_ms,0,blend_radius_m)
    speed_ms = 0.007
    movel([0.104431, -1.350657, -2.591226, -0.770506, 1.570796, 1.675228],accel_mss,speed_ms,0,blend_radius_m)
    movel([0.104261, -1.350893, -2.591069, -0.770427, 1.570796, 1.675057],accel_mss,speed_ms,0,blend_radius_m)
    movel([0.103928, -1.351335, -2.590776, -0.770279, 1.570796, 1.674724],accel_mss,speed_ms,0,blend_radius_m)
    movel([0.103535, -1.351849, -2.590434, -0.770106, 1.570796, 1.674331],accel_mss,speed_ms,0,blend_radius_m)
    movel([0.103125, -1.352380, -2.590080, -0.769929, 1.570796, 1.673921],accel_mss,speed_ms,0,blend_radius_m)
    movel([0.102659, -1.352967, -2.589688, -0.769733, 1.570796, 1.673455],accel_mss,speed_ms,0,blend_radius_m)
    movel([0.102306, -1.353375, -2.589417, -0.769598, 1.570796, 1.673103],accel_mss,speed_ms,0,blend_radius_m)
    movel([0.102040, -1.353644, -2.589237, -0.769508, 1.570796, 1.672837],accel_mss,speed_ms,0,blend_radius_m)
    movel([0.101752, -1.353700, -2.589200, -0.769490, 1.570796, 1.672548],accel_mss,speed_ms,0,blend_radius_m)
    movel([0.101801, -1.353407, -2.589395, -0.769587, 1.570796, 1.672598],accel_mss,speed_ms,0,blend_radius_m)
    movel([0.102838, -1.352207, -2.590195, -0.769987, 1.570796, 1.673635],accel_mss,speed_ms,0,blend_radius_m)
    movel([0.103828, -1.351089, -2.590939, -0.770361, 1.570796, 1.674624],accel_mss,speed_ms,0,blend_radius_m)
    movel([0.104352, -1.350571, -2.591283, -0.770535, 1.570796, 1.675148],accel_mss,speed_ms,0,blend_radius_m)
    movel([0.104721, -1.350245, -2.591499, -0.770645, 1.570796, 1.675517],accel_mss,speed_ms,0,blend_radius_m)
    speed_ms = 0.003
    movel([0.104721, -1.353618, -2.593035, -0.765736, 1.570796, 1.675517],accel_mss,speed_ms,0,blend_radius_m)
    speed_ms = 0.007
    movel([0.104431, -1.354029, -2.592761, -0.765599, 1.570796, 1.675228],accel_mss,speed_ms,0,blend_radius_m)
    movel([0.104261, -1.354264, -2.592604, -0.765521, 1.570796, 1.675057],accel_mss,speed_ms,0,blend_radius_m)
    movel([0.103928, -1.354705, -2.592310, -0.765375, 1.570796, 1.674724],accel_mss,speed_ms,0,blend_radius_m)
    movel([0.103535, -1.355217, -2.591967, -0.765205, 1.570796, 1.674331],accel_mss,speed_ms,0,blend_radius_m)
    movel([0.103125, -1.355748, -2.591612, -0.765029, 1.570796, 1.673921],accel_mss,speed_ms,0,blend_radius_m)
    movel([0.102659, -1.356333, -2.591220, -0.764836, 1.570796, 1.673455],accel_mss,speed_ms,0,blend_radius_m)
    movel([0.102306, -1.356740, -2.590947, -0.764702, 1.570796, 1.673103],accel_mss,speed_ms,0,blend_radius_m)
    movel([0.102040, -1.357008, -2.590767, -0.764614, 1.570796, 1.672837],accel_mss,speed_ms,0,blend_radius_m)
    movel([0.101752, -1.357064, -2.590730, -0.764596, 1.570796, 1.672548],accel_mss,speed_ms,0,blend_radius_m)
    movel([0.101801, -1.356771, -2.590926, -0.764692, 1.570796, 1.672598],accel_mss,speed_ms,0,blend_radius_m)
    movel([0.102838, -1.355574, -2.591728, -0.765087, 1.570796, 1.673635],accel_mss,speed_ms,0,blend_radius_m)
    movel([0.103828, -1.354460, -2.592473, -0.765456, 1.570796, 1.674624],accel_mss,speed_ms,0,blend_radius_m)
    movel([0.104352, -1.353943, -2.592818, -0.765628, 1.570796, 1.675148],accel_mss,speed_ms,0,blend_radius_m)
    movel([0.104721, -1.353618, -2.593035, -0.765736, 1.570796, 1.675517],accel_mss,speed_ms,0,blend_radius_m)
    speed_ms = 0.003
    movel([0.104721, -1.340273, -2.586841, -0.785274, 1.570796, 1.675517],accel_mss,speed_ms,0,blend_radius_m)
    speed_ms = 1.000
    movel([0.104721, -1.314744, -2.574062, -0.823583, 1.570796, 1.675517],accel_mss,speed_ms,0,blend_radius_m)
    movel([0.129209, -1.310300, -2.576848, -0.825241, 1.570796, 1.700005],accel_mss,speed_ms,0,blend_radius_m)
    movel([0.129209, -1.335902, -2.589685, -0.786802, 1.570796, 1.700005],accel_mss,speed_ms,0,blend_radius_m)
    speed_ms = 0.003
    movel([0.129209, -1.345905, -2.594365, -0.772119, 1.570796, 1.700005],accel_mss,speed_ms,0,blend_radius_m)
    speed_ms = 0.007
    movel([0.130130, -1.345778, -2.594448, -0.772163, 1.570796, 1.700926],accel_mss,speed_ms,0,blend_radius_m)
    movel([0.130918, -1.345778, -2.594448, -0.772163, 1.570796, 1.701714],accel_mss,speed_ms,0,blend_radius_m)
    movel([0.131621, -1.345811, -2.594427, -0.772151, 1.570796, 1.702417],accel_mss,speed_ms,0,blend_radius_m)
    movel([0.131927, -1.345942, -2.594340, -0.772106, 1.570796, 1.702724],accel_mss,speed_ms,0,blend_radius_m)
    movel([0.131753, -1.346175, -2.594188, -0.772027, 1.570796, 1.702549],accel_mss,speed_ms,0,blend_radius_m)
    movel([0.131438, -1.346266, -2.594127, -0.771995, 1.570796, 1.702234],accel_mss,speed_ms,0,blend_radius_m)
    movel([0.130444, -1.346251, -2.594137, -0.772001, 1.570796, 1.701240],accel_mss,speed_ms,0,blend_radius_m)
    movel([0.129464, -1.346204, -2.594168, -0.772017, 1.570796, 1.700260],accel_mss,speed_ms,0,blend_radius_m)
    movel([0.129246, -1.346094, -2.594241, -0.772055, 1.570796, 1.700042],accel_mss,speed_ms,0,blend_radius_m)
    speed_ms = 0.003
    movel([0.129209, -1.349289, -2.595908, -0.767192, 1.570796, 1.700005],accel_mss,speed_ms,0,blend_radius_m)
    speed_ms = 0.007
    movel([0.130130, -1.349162, -2.595992, -0.767235, 1.570796, 1.700926],accel_mss,speed_ms,0,blend_radius_m)
    movel([0.130918, -1.349162, -2.595991, -0.767235, 1.570796, 1.701714],accel_mss,speed_ms,0,blend_radius_m)
    movel([0.131621, -1.349195, -2.595970, -0.767224, 1.570796, 1.702417],accel_mss,speed_ms,0,blend_radius_m)
    movel([0.131927, -1.349326, -2.595883, -0.767180, 1.570796, 1.702724],accel_mss,speed_ms,0,blend_radius_m)
    movel([0.131753, -1.349558, -2.595730, -0.767101, 1.570796, 1.702549],accel_mss,speed_ms,0,blend_radius_m)
    movel([0.131438, -1.349649, -2.595670, -0.767070, 1.570796, 1.702234],accel_mss,speed_ms,0,blend_radius_m)
    movel([0.130444, -1.349634, -2.595680, -0.767075, 1.570796, 1.701240],accel_mss,speed_ms,0,blend_radius_m)
    movel([0.129464, -1.349587, -2.595711, -0.767091, 1.570796, 1.700260],accel_mss,speed_ms,0,blend_radius_m)
    movel([0.129246, -1.349477, -2.595784, -0.767128, 1.570796, 1.700042],accel_mss,speed_ms,0,blend_radius_m)
    speed_ms = 0.003
    movel([0.129209, -1.335902, -2.589685, -0.786802, 1.570796, 1.700005],accel_mss,speed_ms,0,blend_radius_m)
    speed_ms = 1.000
    movel([0.129209, -1.310300, -2.576848, -0.825241, 1.570796, 1.700005],accel_mss,speed_ms,0,blend_radius_m)
    movel([0.133372, -1.307920, -2.578330, -0.826139, 1.570796, 1.704169],accel_mss,speed_ms,0,blend_radius_m)
    movel([0.133372, -1.333561, -2.591198, -0.787631, 1.570796, 1.704169],accel_mss,speed_ms,0,blend_radius_m)
    speed_ms = 0.003
    movel([0.133372, -1.343581, -2.595889, -0.772919, 1.570796, 1.704169],accel_mss,speed_ms,0,blend_radius_m)
    speed_ms = 0.007
    movel([0.133523, -1.343804, -2.595743, -0.772842, 1.570796, 1.704320],accel_mss,speed_ms,0,blend_radius_m)
    movel([0.133757, -1.343909, -2.595674, -0.772806, 1.570796, 1.704553],accel_mss,speed_ms,0,blend_radius_m)
    movel([0.133786, -1.344214, -2.595475, -0.772701, 1.570796, 1.704582],accel_mss,speed_ms,0,blend_radius_m)
    movel([0.133733, -1.344526, -2.595270, -0.772593, 1.570796, 1.704530],accel_mss,speed_ms,0,blend_radius_m)
    movel([0.133693, -1.344774, -2.595107, -0.772508, 1.570796, 1.704490],accel_mss,speed_ms,0,blend_radius_m)
    movel([0.133685, -1.345123, -2.594878, -0.772387, 1.570796, 1.704481],accel_mss,speed_ms,0,blend_radius_m)
    movel([0.133764, -1.345308, -2.594757, -0.772324, 1.570796, 1.704561],accel_mss,speed_ms,0,blend_radius_m)
    movel([0.133678, -1.345762, -2.594459, -0.772168, 1.570796, 1.704474],accel_mss,speed_ms,0,blend_radius_m)
    movel([0.133620, -1.346014, -2.594293, -0.772082, 1.570796, 1.704416],accel_mss,speed_ms,0,blend_radius_m)
    movel([0.133584, -1.346401, -2.594039, -0.771949, 1.570796, 1.704380],accel_mss,speed_ms,0,blend_radius_m)
    movel([0.133696, -1.346576, -2.593924, -0.771890, 1.570796, 1.704493],accel_mss,speed_ms,0,blend_radius_m)
    movel([0.133614, -1.347215, -2.593502, -0.771671, 1.570796, 1.704411],accel_mss,speed_ms,0,blend_radius_m)
    movel([0.133501, -1.347865, -2.593074, -0.771450, 1.570796, 1.704297],accel_mss,speed_ms,0,blend_radius_m)
    movel([0.133318, -1.348123, -2.592904, -0.771362, 1.570796, 1.704114],accel_mss,speed_ms,0,blend_radius_m)
    movel([0.133224, -1.348613, -2.592580, -0.771196, 1.570796, 1.704020],accel_mss,speed_ms,0,blend_radius_m)
    movel([0.133196, -1.348926, -2.592373, -0.771090, 1.570796, 1.703993],accel_mss,speed_ms,0,blend_radius_m)
    movel([0.133171, -1.349242, -2.592164, -0.770983, 1.570796, 1.703967],accel_mss,speed_ms,0,blend_radius_m)
    movel([0.133130, -1.349497, -2.591995, -0.770897, 1.570796, 1.703926],accel_mss,speed_ms,0,blend_radius_m)
    movel([0.133029, -1.349737, -2.591836, -0.770816, 1.570796, 1.703825],accel_mss,speed_ms,0,blend_radius_m)
    movel([0.132912, -1.350001, -2.591661, -0.770727, 1.570796, 1.703709],accel_mss,speed_ms,0,blend_radius_m)
    movel([0.132787, -1.350833, -2.591109, -0.770447, 1.570796, 1.703583],accel_mss,speed_ms,0,blend_radius_m)
    movel([0.132241, -1.352571, -2.589953, -0.769865, 1.570796, 1.703037],accel_mss,speed_ms,0,blend_radius_m)
    movel([0.131630, -1.354418, -2.588720, -0.769252, 1.570796, 1.702426],accel_mss,speed_ms,0,blend_radius_m)
    movel([0.131422, -1.354684, -2.588541, -0.769163, 1.570796, 1.702219],accel_mss,speed_ms,0,blend_radius_m)
    movel([0.131217, -1.355020, -2.588316, -0.769053, 1.570796, 1.702013],accel_mss,speed_ms,0,blend_radius_m)
    movel([0.131469, -1.355313, -2.588120, -0.768956, 1.570796, 1.702265],accel_mss,speed_ms,0,blend_radius_m)
    movel([0.131675, -1.355437, -2.588037, -0.768915, 1.570796, 1.702471],accel_mss,speed_ms,0,blend_radius_m)
    movel([0.131656, -1.355707, -2.587856, -0.768826, 1.570796, 1.702453],accel_mss,speed_ms,0,blend_radius_m)
    movel([0.131428, -1.355961, -2.587685, -0.768742, 1.570796, 1.702225],accel_mss,speed_ms,0,blend_radius_m)
    movel([0.131132, -1.356262, -2.587483, -0.768644, 1.570796, 1.701929],accel_mss,speed_ms,0,blend_radius_m)
    movel([0.127085, -1.356793, -2.587126, -0.768469, 1.570796, 1.697882],accel_mss,speed_ms,0,blend_radius_m)
    movel([0.125499, -1.357008, -2.586982, -0.768399, 1.570796, 1.696296],accel_mss,speed_ms,0,blend_radius_m)
    movel([0.124079, -1.357201, -2.586852, -0.768336, 1.570796, 1.694875],accel_mss,speed_ms,0,blend_radius_m)
    movel([0.122882, -1.357368, -2.586740, -0.768282, 1.570796, 1.693678],accel_mss,speed_ms,0,blend_radius_m)
    movel([0.122534, -1.357421, -2.586704, -0.768264, 1.570796, 1.693331],accel_mss,speed_ms,0,blend_radius_m)
    movel([0.122267, -1.357464, -2.586675, -0.768250, 1.570796, 1.693063],accel_mss,speed_ms,0,blend_radius_m)
    movel([0.121847, -1.357524, -2.586635, -0.768230, 1.570796, 1.692643],accel_mss,speed_ms,0,blend_radius_m)
    movel([0.121369, -1.357592, -2.586589, -0.768208, 1.570796, 1.692165],accel_mss,speed_ms,0,blend_radius_m)
    movel([0.120899, -1.357655, -2.586546, -0.768188, 1.570796, 1.691695],accel_mss,speed_ms,0,blend_radius_m)
    movel([0.120401, -1.357724, -2.586500, -0.768165, 1.570796, 1.691197],accel_mss,speed_ms,0,blend_radius_m)
    movel([0.119840, -1.357800, -2.586449, -0.768140, 1.570796, 1.690636],accel_mss,speed_ms,0,blend_radius_m)
    movel([0.119304, -1.357875, -2.586398, -0.768116, 1.570796, 1.690101],accel_mss,speed_ms,0,blend_radius_m)
    movel([0.118887, -1.357934, -2.586358, -0.768097, 1.570796, 1.689683],accel_mss,speed_ms,0,blend_radius_m)
    movel([0.118469, -1.357995, -2.586317, -0.768077, 1.570796, 1.689265],accel_mss,speed_ms,0,blend_radius_m)
    movel([0.117933, -1.358069, -2.586268, -0.768053, 1.570796, 1.688730],accel_mss,speed_ms,0,blend_radius_m)
    movel([0.117372, -1.358148, -2.586214, -0.768027, 1.570796, 1.688169],accel_mss,speed_ms,0,blend_radius_m)
    movel([0.116874, -1.358218, -2.586167, -0.768004, 1.570796, 1.687671],accel_mss,speed_ms,0,blend_radius_m)
    movel([0.114544, -1.358551, -2.585942, -0.767896, 1.570796, 1.685341],accel_mss,speed_ms,0,blend_radius_m)
    movel([0.111844, -1.358958, -2.585668, -0.767764, 1.570796, 1.682641],accel_mss,speed_ms,0,blend_radius_m)
    movel([0.109120, -1.359383, -2.585380, -0.767626, 1.570796, 1.679916],accel_mss,speed_ms,0,blend_radius_m)
    movel([0.108772, -1.359460, -2.585328, -0.767601, 1.570796, 1.679568],accel_mss,speed_ms,0,blend_radius_m)
    movel([0.108514, -1.359224, -2.585488, -0.767677, 1.570796, 1.679311],accel_mss,speed_ms,0,blend_radius_m)
    movel([0.108672, -1.358892, -2.585712, -0.767785, 1.570796, 1.679468],accel_mss,speed_ms,0,blend_radius_m)
    movel([0.108981, -1.358556, -2.585939, -0.767894, 1.570796, 1.679777],accel_mss,speed_ms,0,blend_radius_m)
    movel([0.109311, -1.358296, -2.586114, -0.767979, 1.570796, 1.680107],accel_mss,speed_ms,0,blend_radius_m)
    movel([0.109605, -1.358120, -2.586233, -0.768036, 1.570796, 1.680401],accel_mss,speed_ms,0,blend_radius_m)
    movel([0.109666, -1.357828, -2.586430, -0.768131, 1.570796, 1.680463],accel_mss,speed_ms,0,blend_radius_m)
    movel([0.109470, -1.357719, -2.586503, -0.768167, 1.570796, 1.680266],accel_mss,speed_ms,0,blend_radius_m)
    movel([0.109530, -1.357479, -2.586665, -0.768245, 1.570796, 1.680326],accel_mss,speed_ms,0,blend_radius_m)
    movel([0.109705, -1.357223, -2.586837, -0.768329, 1.570796, 1.680502],accel_mss,speed_ms,0,blend_radius_m)
    movel([0.109652, -1.356857, -2.587083, -0.768449, 1.570796, 1.680449],accel_mss,speed_ms,0,blend_radius_m)
    movel([0.109837, -1.356609, -2.587250, -0.768530, 1.570796, 1.680633],accel_mss,speed_ms,0,blend_radius_m)
    movel([0.109967, -1.356167, -2.587547, -0.768675, 1.570796, 1.680764],accel_mss,speed_ms,0,blend_radius_m)
    movel([0.110006, -1.355882, -2.587738, -0.768768, 1.570796, 1.680802],accel_mss,speed_ms,0,blend_radius_m)
    movel([0.110093, -1.355310, -2.588122, -0.768957, 1.570796, 1.680889],accel_mss,speed_ms,0,blend_radius_m)
    movel([0.110206, -1.354843, -2.588435, -0.769111, 1.570796, 1.681003],accel_mss,speed_ms,0,blend_radius_m)
    movel([0.110408, -1.354229, -2.588846, -0.769314, 1.570796, 1.681205],accel_mss,speed_ms,0,blend_radius_m)
    movel([0.110894, -1.352904, -2.589731, -0.769754, 1.570796, 1.681691],accel_mss,speed_ms,0,blend_radius_m)
    movel([0.111101, -1.352357, -2.590096, -0.769937, 1.570796, 1.681897],accel_mss,speed_ms,0,blend_radius_m)
    movel([0.111293, -1.351885, -2.590410, -0.770094, 1.570796, 1.682089],accel_mss,speed_ms,0,blend_radius_m)
    movel([0.111466, -1.351484, -2.590676, -0.770229, 1.570796, 1.682262],accel_mss,speed_ms,0,blend_radius_m)
    movel([0.111570, -1.351218, -2.590853, -0.770318, 1.570796, 1.682366],accel_mss,speed_ms,0,blend_radius_m)
    movel([0.111744, -1.350968, -2.591019, -0.770402, 1.570796, 1.682540],accel_mss,speed_ms,0,blend_radius_m)
    movel([0.111777, -1.350613, -2.591255, -0.770521, 1.570796, 1.682573],accel_mss,speed_ms,0,blend_radius_m)
    movel([0.112301, -1.349502, -2.591991, -0.770895, 1.570796, 1.683097],accel_mss,speed_ms,0,blend_radius_m)
    movel([0.112851, -1.348413, -2.592712, -0.771264, 1.570796, 1.683647],accel_mss,speed_ms,0,blend_radius_m)
    movel([0.113284, -1.347690, -2.593189, -0.771509, 1.570796, 1.684081],accel_mss,speed_ms,0,blend_radius_m)
    movel([0.113462, -1.347437, -2.593356, -0.771596, 1.570796, 1.684258],accel_mss,speed_ms,0,blend_radius_m)
    movel([0.113667, -1.347170, -2.593532, -0.771687, 1.570796, 1.684463],accel_mss,speed_ms,0,blend_radius_m)
    movel([0.113872, -1.346920, -2.593697, -0.771772, 1.570796, 1.684668],accel_mss,speed_ms,0,blend_radius_m)
    movel([0.114255, -1.346494, -2.593977, -0.771917, 1.570796, 1.685052],accel_mss,speed_ms,0,blend_radius_m)
    movel([0.114419, -1.346139, -2.594211, -0.772039, 1.570796, 1.685216],accel_mss,speed_ms,0,blend_radius_m)
    movel([0.114172, -1.346157, -2.594199, -0.772033, 1.570796, 1.684968],accel_mss,speed_ms,0,blend_radius_m)
    movel([0.113906, -1.346180, -2.594184, -0.772025, 1.570796, 1.684702],accel_mss,speed_ms,0,blend_radius_m)
    movel([0.113638, -1.346105, -2.594234, -0.772051, 1.570796, 1.684434],accel_mss,speed_ms,0,blend_radius_m)
    movel([0.113581, -1.345731, -2.594479, -0.772179, 1.570796, 1.684377],accel_mss,speed_ms,0,blend_radius_m)
    movel([0.113640, -1.345330, -2.594742, -0.772316, 1.570796, 1.684437],accel_mss,speed_ms,0,blend_radius_m)
    movel([0.113813, -1.345065, -2.594916, -0.772408, 1.570796, 1.684609],accel_mss,speed_ms,0,blend_radius_m)
    movel([0.114104, -1.344827, -2.595072, -0.772489, 1.570796, 1.684901],accel_mss,speed_ms,0,blend_radius_m)
    movel([0.114427, -1.344625, -2.595205, -0.772559, 1.570796, 1.685223],accel_mss,speed_ms,0,blend_radius_m)
    movel([0.114780, -1.344455, -2.595316, -0.772617, 1.570796, 1.685576],accel_mss,speed_ms,0,blend_radius_m)
    movel([0.115153, -1.344327, -2.595400, -0.772662, 1.570796, 1.685950],accel_mss,speed_ms,0,blend_radius_m)
    movel([0.115538, -1.344186, -2.595493, -0.772710, 1.570796, 1.686334],accel_mss,speed_ms,0,blend_radius_m)
    movel([0.116178, -1.343789, -2.595752, -0.772847, 1.570796, 1.686974],accel_mss,speed_ms,0,blend_radius_m)
    movel([0.118416, -1.343039, -2.596243, -0.773107, 1.570796, 1.689213],accel_mss,speed_ms,0,blend_radius_m)
    movel([0.120675, -1.342306, -2.596722, -0.773362, 1.570796, 1.691471],accel_mss,speed_ms,0,blend_radius_m)
    movel([0.120996, -1.342326, -2.596708, -0.773355, 1.570796, 1.691792],accel_mss,speed_ms,0,blend_radius_m)
    movel([0.121352, -1.342346, -2.596696, -0.773348, 1.570796, 1.692148],accel_mss,speed_ms,0,blend_radius_m)
    movel([0.121691, -1.342126, -2.596839, -0.773424, 1.570796, 1.692487],accel_mss,speed_ms,0,blend_radius_m)
    movel([0.121589, -1.341884, -2.596996, -0.773508, 1.570796, 1.692385],accel_mss,speed_ms,0,blend_radius_m)
    movel([0.121500, -1.341581, -2.597194, -0.773614, 1.570796, 1.692296],accel_mss,speed_ms,0,blend_radius_m)
    movel([0.121695, -1.341353, -2.597342, -0.773694, 1.570796, 1.692491],accel_mss,speed_ms,0,blend_radius_m)
    movel([0.122038, -1.341103, -2.597505, -0.773781, 1.570796, 1.692835],accel_mss,speed_ms,0,blend_radius_m)
    movel([0.122298, -1.340917, -2.597626, -0.773846, 1.570796, 1.693094],accel_mss,speed_ms,0,blend_radius_m)
    movel([0.122428, -1.340654, -2.597797, -0.773938, 1.570796, 1.693224],accel_mss,speed_ms,0,blend_radius_m)
    movel([0.122134, -1.340648, -2.597801, -0.773940, 1.570796, 1.692931],accel_mss,speed_ms,0,blend_radius_m)
    movel([0.121865, -1.340652, -2.597798, -0.773938, 1.570796, 1.692661],accel_mss,speed_ms,0,blend_radius_m)
    movel([0.121926, -1.340137, -2.598133, -0.774119, 1.570796, 1.692722],accel_mss,speed_ms,0,blend_radius_m)
    movel([0.122108, -1.339570, -2.598501, -0.774318, 1.570796, 1.692904],accel_mss,speed_ms,0,blend_radius_m)
    movel([0.122198, -1.339304, -2.598673, -0.774411, 1.570796, 1.692994],accel_mss,speed_ms,0,blend_radius_m)
    movel([0.122277, -1.339057, -2.598834, -0.774498, 1.570796, 1.693074],accel_mss,speed_ms,0,blend_radius_m)
    movel([0.122367, -1.338753, -2.599030, -0.774605, 1.570796, 1.693164],accel_mss,speed_ms,0,blend_radius_m)
    movel([0.122577, -1.338442, -2.599232, -0.774715, 1.570796, 1.693373],accel_mss,speed_ms,0,blend_radius_m)
    movel([0.122789, -1.338186, -2.599397, -0.774806, 1.570796, 1.693585],accel_mss,speed_ms,0,blend_radius_m)
    movel([0.123034, -1.337910, -2.599576, -0.774903, 1.570796, 1.693831],accel_mss,speed_ms,0,blend_radius_m)
    movel([0.123671, -1.337217, -2.600024, -0.775149, 1.570796, 1.694467],accel_mss,speed_ms,0,blend_radius_m)
    movel([0.124629, -1.337021, -2.600150, -0.775218, 1.570796, 1.695426],accel_mss,speed_ms,0,blend_radius_m)
    movel([0.125882, -1.336797, -2.600295, -0.775298, 1.570796, 1.696678],accel_mss,speed_ms,0,blend_radius_m)
    movel([0.127200, -1.336622, -2.600407, -0.775360, 1.570796, 1.697996],accel_mss,speed_ms,0,blend_radius_m)
    movel([0.128376, -1.336509, -2.600480, -0.775400, 1.570796, 1.699172],accel_mss,speed_ms,0,blend_radius_m)
    movel([0.128803, -1.336554, -2.600451, -0.775384, 1.570796, 1.699599],accel_mss,speed_ms,0,blend_radius_m)
    movel([0.129089, -1.336680, -2.600370, -0.775339, 1.570796, 1.699886],accel_mss,speed_ms,0,blend_radius_m)
    movel([0.129309, -1.336847, -2.600262, -0.775280, 1.570796, 1.700106],accel_mss,speed_ms,0,blend_radius_m)
    movel([0.129435, -1.337023, -2.600149, -0.775218, 1.570796, 1.700231],accel_mss,speed_ms,0,blend_radius_m)
    movel([0.129396, -1.337284, -2.599980, -0.775125, 1.570796, 1.700193],accel_mss,speed_ms,0,blend_radius_m)
    movel([0.129524, -1.337460, -2.599866, -0.775062, 1.570796, 1.700320],accel_mss,speed_ms,0,blend_radius_m)
    movel([0.129472, -1.337779, -2.599661, -0.774950, 1.570796, 1.700269],accel_mss,speed_ms,0,blend_radius_m)
    movel([0.129264, -1.338017, -2.599507, -0.774865, 1.570796, 1.700060],accel_mss,speed_ms,0,blend_radius_m)
    movel([0.129247, -1.338303, -2.599322, -0.774764, 1.570796, 1.700043],accel_mss,speed_ms,0,blend_radius_m)
    movel([0.129226, -1.338701, -2.599064, -0.774624, 1.570796, 1.700023],accel_mss,speed_ms,0,blend_radius_m)
    movel([0.129118, -1.339164, -2.598765, -0.774461, 1.570796, 1.699915],accel_mss,speed_ms,0,blend_radius_m)
    movel([0.128966, -1.339555, -2.598510, -0.774323, 1.570796, 1.699762],accel_mss,speed_ms,0,blend_radius_m)
    movel([0.128664, -1.339692, -2.598422, -0.774275, 1.570796, 1.699461],accel_mss,speed_ms,0,blend_radius_m)
    movel([0.128382, -1.339893, -2.598292, -0.774205, 1.570796, 1.699178],accel_mss,speed_ms,0,blend_radius_m)
    movel([0.128379, -1.340190, -2.598099, -0.774100, 1.570796, 1.699175],accel_mss,speed_ms,0,blend_radius_m)
    movel([0.128483, -1.340437, -2.597939, -0.774014, 1.570796, 1.699279],accel_mss,speed_ms,0,blend_radius_m)
    movel([0.128519, -1.340727, -2.597750, -0.773912, 1.570796, 1.699315],accel_mss,speed_ms,0,blend_radius_m)
    movel([0.128237, -1.340991, -2.597578, -0.773820, 1.570796, 1.699033],accel_mss,speed_ms,0,blend_radius_m)
    movel([0.128151, -1.341286, -2.597386, -0.773717, 1.570796, 1.698948],accel_mss,speed_ms,0,blend_radius_m)
    movel([0.128545, -1.341249, -2.597410, -0.773730, 1.570796, 1.699342],accel_mss,speed_ms,0,blend_radius_m)
    movel([0.129417, -1.341135, -2.597484, -0.773769, 1.570796, 1.700213],accel_mss,speed_ms,0,blend_radius_m)
    movel([0.130216, -1.341116, -2.597497, -0.773776, 1.570796, 1.701013],accel_mss,speed_ms,0,blend_radius_m)
    movel([0.130962, -1.341141, -2.597481, -0.773768, 1.570796, 1.701758],accel_mss,speed_ms,0,blend_radius_m)
    movel([0.131239, -1.341229, -2.597423, -0.773737, 1.570796, 1.702036],accel_mss,speed_ms,0,blend_radius_m)
    movel([0.131699, -1.341255, -2.597406, -0.773728, 1.570796, 1.702495],accel_mss,speed_ms,0,blend_radius_m)
    movel([0.132047, -1.341071, -2.597526, -0.773792, 1.570796, 1.702843],accel_mss,speed_ms,0,blend_radius_m)
    movel([0.131918, -1.340895, -2.597641, -0.773854, 1.570796, 1.702714],accel_mss,speed_ms,0,blend_radius_m)
    movel([0.131651, -1.340703, -2.597765, -0.773921, 1.570796, 1.702447],accel_mss,speed_ms,0,blend_radius_m)
    movel([0.132106, -1.340258, -2.598054, -0.774076, 1.570796, 1.702902],accel_mss,speed_ms,0,blend_radius_m)
    movel([0.132430, -1.340052, -2.598188, -0.774149, 1.570796, 1.703227],accel_mss,speed_ms,0,blend_radius_m)
    movel([0.132572, -1.339811, -2.598345, -0.774233, 1.570796, 1.703368],accel_mss,speed_ms,0,blend_radius_m)
    movel([0.132296, -1.339674, -2.598433, -0.774281, 1.570796, 1.703093],accel_mss,speed_ms,0,blend_radius_m)
    movel([0.132431, -1.339196, -2.598743, -0.774449, 1.570796, 1.703227],accel_mss,speed_ms,0,blend_radius_m)
    movel([0.132665, -1.338954, -2.598900, -0.774535, 1.570796, 1.703462],accel_mss,speed_ms,0,blend_radius_m)
    movel([0.133142, -1.338621, -2.599116, -0.774652, 1.570796, 1.703938],accel_mss,speed_ms,0,blend_radius_m)
    movel([0.133515, -1.338463, -2.599218, -0.774708, 1.570796, 1.704311],accel_mss,speed_ms,0,blend_radius_m)
    movel([0.133874, -1.338443, -2.599231, -0.774715, 1.570796, 1.704671],accel_mss,speed_ms,0,blend_radius_m)
    movel([0.134312, -1.338556, -2.599158, -0.774675, 1.570796, 1.705108],accel_mss,speed_ms,0,blend_radius_m)
    movel([0.134537, -1.338645, -2.599101, -0.774644, 1.570796, 1.705333],accel_mss,speed_ms,0,blend_radius_m)
    movel([0.134724, -1.338732, -2.599044, -0.774613, 1.570796, 1.705520],accel_mss,speed_ms,0,blend_radius_m)
    movel([0.134889, -1.338852, -2.598966, -0.774570, 1.570796, 1.705685],accel_mss,speed_ms,0,blend_radius_m)
    movel([0.135058, -1.339061, -2.598831, -0.774497, 1.570796, 1.705854],accel_mss,speed_ms,0,blend_radius_m)
    movel([0.135120, -1.339390, -2.598618, -0.774381, 1.570796, 1.705917],accel_mss,speed_ms,0,blend_radius_m)
    movel([0.134596, -1.339904, -2.598284, -0.774201, 1.570796, 1.705392],accel_mss,speed_ms,0,blend_radius_m)
    movel([0.134152, -1.340236, -2.598069, -0.774084, 1.570796, 1.704948],accel_mss,speed_ms,0,blend_radius_m)
    movel([0.134394, -1.340409, -2.597957, -0.774024, 1.570796, 1.705190],accel_mss,speed_ms,0,blend_radius_m)
    movel([0.134638, -1.340583, -2.597843, -0.773963, 1.570796, 1.705434],accel_mss,speed_ms,0,blend_radius_m)
    movel([0.134303, -1.340887, -2.597646, -0.773856, 1.570796, 1.705100],accel_mss,speed_ms,0,blend_radius_m)
    movel([0.133995, -1.341122, -2.597493, -0.773774, 1.570796, 1.704791],accel_mss,speed_ms,0,blend_radius_m)
    movel([0.133724, -1.341260, -2.597403, -0.773726, 1.570796, 1.704520],accel_mss,speed_ms,0,blend_radius_m)
    movel([0.133806, -1.341542, -2.597219, -0.773628, 1.570796, 1.704602],accel_mss,speed_ms,0,blend_radius_m)
    movel([0.134102, -1.341551, -2.597214, -0.773625, 1.570796, 1.704899],accel_mss,speed_ms,0,blend_radius_m)
    movel([0.134405, -1.341598, -2.597183, -0.773608, 1.570796, 1.705202],accel_mss,speed_ms,0,blend_radius_m)
    movel([0.134632, -1.341752, -2.597083, -0.773554, 1.570796, 1.705428],accel_mss,speed_ms,0,blend_radius_m)
    movel([0.134781, -1.341889, -2.596993, -0.773507, 1.570796, 1.705577],accel_mss,speed_ms,0,blend_radius_m)
    movel([0.134990, -1.341997, -2.596923, -0.773469, 1.570796, 1.705786],accel_mss,speed_ms,0,blend_radius_m)
    movel([0.134941, -1.342299, -2.596726, -0.773364, 1.570796, 1.705737],accel_mss,speed_ms,0,blend_radius_m)
    movel([0.134735, -1.342517, -2.596584, -0.773288, 1.570796, 1.705532],accel_mss,speed_ms,0,blend_radius_m)
    movel([0.134593, -1.342795, -2.596402, -0.773192, 1.570796, 1.705389],accel_mss,speed_ms,0,blend_radius_m)
    movel([0.134351, -1.343086, -2.596212, -0.773091, 1.570796, 1.705148],accel_mss,speed_ms,0,blend_radius_m)
    movel([0.134008, -1.343305, -2.596069, -0.773015, 1.570796, 1.704805],accel_mss,speed_ms,0,blend_radius_m)
    movel([0.133511, -1.343459, -2.595968, -0.772961, 1.570796, 1.704307],accel_mss,speed_ms,0,blend_radius_m)
    speed_ms = 0.003
    movel([0.133372, -1.346971, -2.597436, -0.767983, 1.570796, 1.704169],accel_mss,speed_ms,0,blend_radius_m)
    speed_ms = 0.007
    movel([0.133523, -1.347193, -2.597289, -0.767907, 1.570796, 1.704320],accel_mss,speed_ms,0,blend_radius_m)
    movel([0.133757, -1.347298, -2.597220, -0.767871, 1.570796, 1.704553],accel_mss,speed_ms,0,blend_radius_m)
    movel([0.133786, -1.347602, -2.597020, -0.767767, 1.570796, 1.704582],accel_mss,speed_ms,0,blend_radius_m)
    movel([0.133733, -1.347914, -2.596815, -0.767660, 1.570796, 1.704530],accel_mss,speed_ms,0,blend_radius_m)
    movel([0.133693, -1.348161, -2.596652, -0.767576, 1.570796, 1.704490],accel_mss,speed_ms,0,blend_radius_m)
    movel([0.133685, -1.348509, -2.596422, -0.767457, 1.570796, 1.704481],accel_mss,speed_ms,0,blend_radius_m)
    movel([0.133764, -1.348693, -2.596301, -0.767395, 1.570796, 1.704561],accel_mss,speed_ms,0,blend_radius_m)
    movel([0.133678, -1.349146, -2.596002, -0.767241, 1.570796, 1.704474],accel_mss,speed_ms,0,blend_radius_m)
    movel([0.133620, -1.349397, -2.595836, -0.767156, 1.570796, 1.704416],accel_mss,speed_ms,0,blend_radius_m)
    movel([0.133584, -1.349783, -2.595581, -0.767025, 1.570796, 1.704380],accel_mss,speed_ms,0,blend_radius_m)
    movel([0.133696, -1.349958, -2.595466, -0.766966, 1.570796, 1.704493],accel_mss,speed_ms,0,blend_radius_m)
    movel([0.133614, -1.350596, -2.595043, -0.766750, 1.570796, 1.704411],accel_mss,speed_ms,0,blend_radius_m)
    movel([0.133501, -1.351244, -2.594614, -0.766532, 1.570796, 1.704297],accel_mss,speed_ms,0,blend_radius_m)
    movel([0.133318, -1.351501, -2.594443, -0.766445, 1.570796, 1.704114],accel_mss,speed_ms,0,blend_radius_m)
    movel([0.133224, -1.351989, -2.594119, -0.766281, 1.570796, 1.704020],accel_mss,speed_ms,0,blend_radius_m)
    movel([0.133196, -1.352302, -2.593911, -0.766176, 1.570796, 1.703993],accel_mss,speed_ms,0,blend_radius_m)
    movel([0.133171, -1.352618, -2.593701, -0.766070, 1.570796, 1.703967],accel_mss,speed_ms,0,blend_radius_m)
    movel([0.133130, -1.352872, -2.593532, -0.765985, 1.570796, 1.703926],accel_mss,speed_ms,0,blend_radius_m)
    movel([0.133029, -1.353111, -2.593372, -0.765905, 1.570796, 1.703825],accel_mss,speed_ms,0,blend_radius_m)
    movel([0.132912, -1.353375, -2.593197, -0.765817, 1.570796, 1.703709],accel_mss,speed_ms,0,blend_radius_m)
    movel([0.132787, -1.354205, -2.592644, -0.765541, 1.570796, 1.703583],accel_mss,speed_ms,0,blend_radius_m)
    movel([0.132241, -1.355938, -2.591485, -0.764967, 1.570796, 1.703037],accel_mss,speed_ms,0,blend_radius_m)
    movel([0.131630, -1.357780, -2.590248, -0.764361, 1.570796, 1.702426],accel_mss,speed_ms,0,blend_radius_m)
    movel([0.131422, -1.358046, -2.590069, -0.764274, 1.570796, 1.702219],accel_mss,speed_ms,0,blend_radius_m)
    movel([0.131217, -1.358381, -2.589844, -0.764164, 1.570796, 1.702013],accel_mss,speed_ms,0,blend_radius_m)
    movel([0.131469, -1.358672, -2.589647, -0.764069, 1.570796, 1.702265],accel_mss,speed_ms,0,blend_radius_m)
    movel([0.131675, -1.358796, -2.589564, -0.764029, 1.570796, 1.702471],accel_mss,speed_ms,0,blend_radius_m)
    movel([0.131656, -1.359066, -2.589382, -0.763941, 1.570796, 1.702453],accel_mss,speed_ms,0,blend_radius_m)
    movel([0.131428, -1.359319, -2.589211, -0.763858, 1.570796, 1.702225],accel_mss,speed_ms,0,blend_radius_m)
    movel([0.131132, -1.359619, -2.589009, -0.763761, 1.570796, 1.701929],accel_mss,speed_ms,0,blend_radius_m)
    movel([0.127085, -1.360149, -2.588651, -0.763589, 1.570796, 1.697882],accel_mss,speed_ms,0,blend_radius_m)
    movel([0.125499, -1.360363, -2.588507, -0.763519, 1.570796, 1.696296],accel_mss,speed_ms,0,blend_radius_m)
    movel([0.124079, -1.360556, -2.588376, -0.763457, 1.570796, 1.694875],accel_mss,speed_ms,0,blend_radius_m)
    movel([0.122882, -1.360722, -2.588264, -0.763403, 1.570796, 1.693678],accel_mss,speed_ms,0,blend_radius_m)
    movel([0.122534, -1.360775, -2.588228, -0.763386, 1.570796, 1.693331],accel_mss,speed_ms,0,blend_radius_m)
    movel([0.122267, -1.360818, -2.588199, -0.763372, 1.570796, 1.693063],accel_mss,speed_ms,0,blend_radius_m)
    movel([0.121847, -1.360878, -2.588158, -0.763353, 1.570796, 1.692643],accel_mss,speed_ms,0,blend_radius_m)
    movel([0.121369, -1.360945, -2.588113, -0.763331, 1.570796, 1.692165],accel_mss,speed_ms,0,blend_radius_m)
    movel([0.120899, -1.361009, -2.588070, -0.763311, 1.570796, 1.691695],accel_mss,speed_ms,0,blend_radius_m)
    movel([0.120401, -1.361077, -2.588023, -0.763288, 1.570796, 1.691197],accel_mss,speed_ms,0,blend_radius_m)
    movel([0.119840, -1.361153, -2.587972, -0.763264, 1.570796, 1.690636],accel_mss,speed_ms,0,blend_radius_m)
    movel([0.119304, -1.361228, -2.587921, -0.763240, 1.570796, 1.690101],accel_mss,speed_ms,0,blend_radius_m)
    movel([0.118887, -1.361287, -2.587881, -0.763221, 1.570796, 1.689683],accel_mss,speed_ms,0,blend_radius_m)
    movel([0.118469, -1.361347, -2.587840, -0.763201, 1.570796, 1.689265],accel_mss,speed_ms,0,blend_radius_m)
    movel([0.117933, -1.361421, -2.587790, -0.763178, 1.570796, 1.688730],accel_mss,speed_ms,0,blend_radius_m)
    movel([0.117372, -1.361500, -2.587737, -0.763152, 1.570796, 1.688169],accel_mss,speed_ms,0,blend_radius_m)
    movel([0.116874, -1.361570, -2.587689, -0.763129, 1.570796, 1.687671],accel_mss,speed_ms,0,blend_radius_m)
    movel([0.114544, -1.361902, -2.587464, -0.763022, 1.570796, 1.685341],accel_mss,speed_ms,0,blend_radius_m)
    movel([0.111844, -1.362308, -2.587189, -0.762892, 1.570796, 1.682641],accel_mss,speed_ms,0,blend_radius_m)
    movel([0.109120, -1.362733, -2.586901, -0.762756, 1.570796, 1.679916],accel_mss,speed_ms,0,blend_radius_m)
    movel([0.108772, -1.362809, -2.586848, -0.762731, 1.570796, 1.679568],accel_mss,speed_ms,0,blend_radius_m)
    movel([0.108514, -1.362574, -2.587008, -0.762807, 1.570796, 1.679311],accel_mss,speed_ms,0,blend_radius_m)
    movel([0.108672, -1.362243, -2.587233, -0.762913, 1.570796, 1.679468],accel_mss,speed_ms,0,blend_radius_m)
    movel([0.108981, -1.361907, -2.587461, -0.763021, 1.570796, 1.679777],accel_mss,speed_ms,0,blend_radius_m)
    movel([0.109311, -1.361648, -2.587636, -0.763104, 1.570796, 1.680107],accel_mss,speed_ms,0,blend_radius_m)
    movel([0.109605, -1.361472, -2.587756, -0.763161, 1.570796, 1.680401],accel_mss,speed_ms,0,blend_radius_m)
    movel([0.109666, -1.361181, -2.587953, -0.763255, 1.570796, 1.680463],accel_mss,speed_ms,0,blend_radius_m)
    movel([0.109470, -1.361072, -2.588027, -0.763290, 1.570796, 1.680266],accel_mss,speed_ms,0,blend_radius_m)
    movel([0.109530, -1.360833, -2.588189, -0.763367, 1.570796, 1.680326],accel_mss,speed_ms,0,blend_radius_m)
    movel([0.109705, -1.360578, -2.588361, -0.763450, 1.570796, 1.680502],accel_mss,speed_ms,0,blend_radius_m)
    movel([0.109652, -1.360212, -2.588608, -0.763568, 1.570796, 1.680449],accel_mss,speed_ms,0,blend_radius_m)
    movel([0.109837, -1.359966, -2.588775, -0.763648, 1.570796, 1.680633],accel_mss,speed_ms,0,blend_radius_m)
    movel([0.109967, -1.359524, -2.589073, -0.763792, 1.570796, 1.680764],accel_mss,speed_ms,0,blend_radius_m)
    movel([0.110006, -1.359241, -2.589264, -0.763884, 1.570796, 1.680802],accel_mss,speed_ms,0,blend_radius_m)
    movel([0.110093, -1.358670, -2.589649, -0.764070, 1.570796, 1.680889],accel_mss,speed_ms,0,blend_radius_m)
    movel([0.110206, -1.358204, -2.589963, -0.764222, 1.570796, 1.681003],accel_mss,speed_ms,0,blend_radius_m)
    movel([0.110408, -1.357592, -2.590375, -0.764422, 1.570796, 1.681205],accel_mss,speed_ms,0,blend_radius_m)
    movel([0.110894, -1.356270, -2.591262, -0.764857, 1.570796, 1.681691],accel_mss,speed_ms,0,blend_radius_m)
    movel([0.111101, -1.355724, -2.591628, -0.765037, 1.570796, 1.681897],accel_mss,speed_ms,0,blend_radius_m)
    movel([0.111293, -1.355253, -2.591943, -0.765193, 1.570796, 1.682089],accel_mss,speed_ms,0,blend_radius_m)
    movel([0.111466, -1.354854, -2.592210, -0.765325, 1.570796, 1.682262],accel_mss,speed_ms,0,blend_radius_m)
    movel([0.111570, -1.354589, -2.592387, -0.765413, 1.570796, 1.682366],accel_mss,speed_ms,0,blend_radius_m)
    movel([0.111744, -1.354339, -2.592554, -0.765496, 1.570796, 1.682540],accel_mss,speed_ms,0,blend_radius_m)
    movel([0.111777, -1.353985, -2.592790, -0.765614, 1.570796, 1.682573],accel_mss,speed_ms,0,blend_radius_m)
    movel([0.112301, -1.352877, -2.593529, -0.765984, 1.570796, 1.683097],accel_mss,speed_ms,0,blend_radius_m)
    movel([0.112851, -1.351791, -2.594251, -0.766348, 1.570796, 1.683647],accel_mss,speed_ms,0,blend_radius_m)
    movel([0.113284, -1.351070, -2.594729, -0.766590, 1.570796, 1.684081],accel_mss,speed_ms,0,blend_radius_m)
    movel([0.113462, -1.350817, -2.594896, -0.766675, 1.570796, 1.684258],accel_mss,speed_ms,0,blend_radius_m)
    movel([0.113667, -1.350551, -2.595073, -0.766765, 1.570796, 1.684463],accel_mss,speed_ms,0,blend_radius_m)
    movel([0.113872, -1.350302, -2.595238, -0.766849, 1.570796, 1.684668],accel_mss,speed_ms,0,blend_radius_m)
    movel([0.114255, -1.349877, -2.595519, -0.766993, 1.570796, 1.685052],accel_mss,speed_ms,0,blend_radius_m)
    movel([0.114419, -1.349522, -2.595753, -0.767113, 1.570796, 1.685216],accel_mss,speed_ms,0,blend_radius_m)
    movel([0.114172, -1.349540, -2.595742, -0.767107, 1.570796, 1.684968],accel_mss,speed_ms,0,blend_radius_m)
    movel([0.113906, -1.349563, -2.595727, -0.767099, 1.570796, 1.684702],accel_mss,speed_ms,0,blend_radius_m)
    movel([0.113638, -1.349488, -2.595776, -0.767125, 1.570796, 1.684434],accel_mss,speed_ms,0,blend_radius_m)
    movel([0.113581, -1.349115, -2.596022, -0.767251, 1.570796, 1.684377],accel_mss,speed_ms,0,blend_radius_m)
    movel([0.113640, -1.348716, -2.596286, -0.767387, 1.570796, 1.684437],accel_mss,speed_ms,0,blend_radius_m)
    movel([0.113813, -1.348451, -2.596461, -0.767477, 1.570796, 1.684609],accel_mss,speed_ms,0,blend_radius_m)
    movel([0.114104, -1.348214, -2.596617, -0.767558, 1.570796, 1.684901],accel_mss,speed_ms,0,blend_radius_m)
    movel([0.114427, -1.348012, -2.596750, -0.767627, 1.570796, 1.685223],accel_mss,speed_ms,0,blend_radius_m)
    movel([0.114780, -1.347843, -2.596862, -0.767685, 1.570796, 1.685576],accel_mss,speed_ms,0,blend_radius_m)
    movel([0.115153, -1.347715, -2.596946, -0.767728, 1.570796, 1.685950],accel_mss,speed_ms,0,blend_radius_m)
    movel([0.115538, -1.347574, -2.597038, -0.767776, 1.570796, 1.686334],accel_mss,speed_ms,0,blend_radius_m)
    movel([0.116178, -1.347179, -2.597299, -0.767912, 1.570796, 1.686974],accel_mss,speed_ms,0,blend_radius_m)
    movel([0.118416, -1.346430, -2.597791, -0.768168, 1.570796, 1.689213],accel_mss,speed_ms,0,blend_radius_m)
    movel([0.120675, -1.345699, -2.598271, -0.768420, 1.570796, 1.691471],accel_mss,speed_ms,0,blend_radius_m)
    movel([0.120996, -1.345719, -2.598257, -0.768413, 1.570796, 1.691792],accel_mss,speed_ms,0,blend_radius_m)
    movel([0.121352, -1.345738, -2.598245, -0.768406, 1.570796, 1.692148],accel_mss,speed_ms,0,blend_radius_m)
    movel([0.121691, -1.345520, -2.598388, -0.768481, 1.570796, 1.692487],accel_mss,speed_ms,0,blend_radius_m)
    movel([0.121589, -1.345278, -2.598546, -0.768565, 1.570796, 1.692385],accel_mss,speed_ms,0,blend_radius_m)
    movel([0.121500, -1.344976, -2.598744, -0.768669, 1.570796, 1.692296],accel_mss,speed_ms,0,blend_radius_m)
    movel([0.121695, -1.344748, -2.598893, -0.768748, 1.570796, 1.692491],accel_mss,speed_ms,0,blend_radius_m)
    movel([0.122038, -1.344499, -2.599056, -0.768834, 1.570796, 1.692835],accel_mss,speed_ms,0,blend_radius_m)
    movel([0.122298, -1.344313, -2.599178, -0.768898, 1.570796, 1.693094],accel_mss,speed_ms,0,blend_radius_m)
    movel([0.122428, -1.344051, -2.599349, -0.768989, 1.570796, 1.693224],accel_mss,speed_ms,0,blend_radius_m)
    movel([0.122134, -1.344045, -2.599353, -0.768991, 1.570796, 1.692931],accel_mss,speed_ms,0,blend_radius_m)
    movel([0.121865, -1.344049, -2.599350, -0.768989, 1.570796, 1.692661],accel_mss,speed_ms,0,blend_radius_m)
    movel([0.121926, -1.343536, -2.599686, -0.769168, 1.570796, 1.692722],accel_mss,speed_ms,0,blend_radius_m)
    movel([0.122108, -1.342970, -2.600055, -0.769365, 1.570796, 1.692904],accel_mss,speed_ms,0,blend_radius_m)
    movel([0.122198, -1.342705, -2.600227, -0.769457, 1.570796, 1.692994],accel_mss,speed_ms,0,blend_radius_m)
    movel([0.122277, -1.342458, -2.600388, -0.769543, 1.570796, 1.693074],accel_mss,speed_ms,0,blend_radius_m)
    movel([0.122367, -1.342155, -2.600585, -0.769649, 1.570796, 1.693164],accel_mss,speed_ms,0,blend_radius_m)
    movel([0.122577, -1.341845, -2.600787, -0.769757, 1.570796, 1.693373],accel_mss,speed_ms,0,blend_radius_m)
    movel([0.122789, -1.341589, -2.600953, -0.769846, 1.570796, 1.693585],accel_mss,speed_ms,0,blend_radius_m)
    movel([0.123034, -1.341314, -2.601133, -0.769943, 1.570796, 1.693831],accel_mss,speed_ms,0,blend_radius_m)
    movel([0.123671, -1.340622, -2.601581, -0.770185, 1.570796, 1.694467],accel_mss,speed_ms,0,blend_radius_m)
    movel([0.124629, -1.340427, -2.601708, -0.770254, 1.570796, 1.695426],accel_mss,speed_ms,0,blend_radius_m)
    movel([0.125882, -1.340203, -2.601853, -0.770333, 1.570796, 1.696678],accel_mss,speed_ms,0,blend_radius_m)
    movel([0.127200, -1.340030, -2.601965, -0.770394, 1.570796, 1.697996],accel_mss,speed_ms,0,blend_radius_m)
    movel([0.128376, -1.339917, -2.602039, -0.770434, 1.570796, 1.699172],accel_mss,speed_ms,0,blend_radius_m)
    movel([0.128803, -1.339961, -2.602010, -0.770418, 1.570796, 1.699599],accel_mss,speed_ms,0,blend_radius_m)
    movel([0.129089, -1.340087, -2.601928, -0.770374, 1.570796, 1.699886],accel_mss,speed_ms,0,blend_radius_m)
    movel([0.129309, -1.340254, -2.601820, -0.770315, 1.570796, 1.700106],accel_mss,speed_ms,0,blend_radius_m)
    movel([0.129435, -1.340429, -2.601707, -0.770253, 1.570796, 1.700231],accel_mss,speed_ms,0,blend_radius_m)
    movel([0.129396, -1.340689, -2.601538, -0.770162, 1.570796, 1.700193],accel_mss,speed_ms,0,blend_radius_m)
    movel([0.129524, -1.340866, -2.601423, -0.770100, 1.570796, 1.700320],accel_mss,speed_ms,0,blend_radius_m)
    movel([0.129472, -1.341183, -2.601217, -0.769989, 1.570796, 1.700269],accel_mss,speed_ms,0,blend_radius_m)
    movel([0.129264, -1.341421, -2.601063, -0.769905, 1.570796, 1.700060],accel_mss,speed_ms,0,blend_radius_m)
    movel([0.129247, -1.341706, -2.600878, -0.769806, 1.570796, 1.700043],accel_mss,speed_ms,0,blend_radius_m)
    movel([0.129226, -1.342103, -2.600619, -0.769667, 1.570796, 1.700023],accel_mss,speed_ms,0,blend_radius_m)
    movel([0.129118, -1.342564, -2.600319, -0.769506, 1.570796, 1.699915],accel_mss,speed_ms,0,blend_radius_m)
    movel([0.128966, -1.342955, -2.600064, -0.769370, 1.570796, 1.699762],accel_mss,speed_ms,0,blend_radius_m)
    movel([0.128664, -1.343092, -2.599975, -0.769322, 1.570796, 1.699461],accel_mss,speed_ms,0,blend_radius_m)
    movel([0.128382, -1.343292, -2.599845, -0.769252, 1.570796, 1.699178],accel_mss,speed_ms,0,blend_radius_m)
    movel([0.128379, -1.343588, -2.599652, -0.769150, 1.570796, 1.699175],accel_mss,speed_ms,0,blend_radius_m)
    movel([0.128483, -1.343834, -2.599491, -0.769064, 1.570796, 1.699279],accel_mss,speed_ms,0,blend_radius_m)
    movel([0.128519, -1.344124, -2.599301, -0.768964, 1.570796, 1.699315],accel_mss,speed_ms,0,blend_radius_m)
    movel([0.128237, -1.344388, -2.599129, -0.768872, 1.570796, 1.699033],accel_mss,speed_ms,0,blend_radius_m)
    movel([0.128151, -1.344682, -2.598937, -0.768771, 1.570796, 1.698948],accel_mss,speed_ms,0,blend_radius_m)
    movel([0.128545, -1.344644, -2.598961, -0.768784, 1.570796, 1.699342],accel_mss,speed_ms,0,blend_radius_m)
    movel([0.129417, -1.344531, -2.599035, -0.768823, 1.570796, 1.700213],accel_mss,speed_ms,0,blend_radius_m)
    movel([0.130216, -1.344512, -2.599048, -0.768829, 1.570796, 1.701013],accel_mss,speed_ms,0,blend_radius_m)
    movel([0.130962, -1.344536, -2.599032, -0.768821, 1.570796, 1.701758],accel_mss,speed_ms,0,blend_radius_m)
    movel([0.131239, -1.344625, -2.598974, -0.768790, 1.570796, 1.702036],accel_mss,speed_ms,0,blend_radius_m)
    movel([0.131699, -1.344650, -2.598957, -0.768781, 1.570796, 1.702495],accel_mss,speed_ms,0,blend_radius_m)
    movel([0.132047, -1.344467, -2.599077, -0.768845, 1.570796, 1.702843],accel_mss,speed_ms,0,blend_radius_m)
    movel([0.131918, -1.344291, -2.599192, -0.768906, 1.570796, 1.702714],accel_mss,speed_ms,0,blend_radius_m)
    movel([0.131651, -1.344100, -2.599317, -0.768972, 1.570796, 1.702447],accel_mss,speed_ms,0,blend_radius_m)
    movel([0.132106, -1.343657, -2.599607, -0.769126, 1.570796, 1.702902],accel_mss,speed_ms,0,blend_radius_m)
    movel([0.132430, -1.343451, -2.599741, -0.769197, 1.570796, 1.703227],accel_mss,speed_ms,0,blend_radius_m)
    movel([0.132572, -1.343210, -2.599898, -0.769281, 1.570796, 1.703368],accel_mss,speed_ms,0,blend_radius_m)
    movel([0.132296, -1.343074, -2.599987, -0.769328, 1.570796, 1.703093],accel_mss,speed_ms,0,blend_radius_m)
    movel([0.132431, -1.342597, -2.600298, -0.769494, 1.570796, 1.703227],accel_mss,speed_ms,0,blend_radius_m)
    movel([0.132665, -1.342355, -2.600455, -0.769579, 1.570796, 1.703462],accel_mss,speed_ms,0,blend_radius_m)
    movel([0.133142, -1.342023, -2.600671, -0.769695, 1.570796, 1.703938],accel_mss,speed_ms,0,blend_radius_m)
    movel([0.133515, -1.341866, -2.600774, -0.769750, 1.570796, 1.704311],accel_mss,speed_ms,0,blend_radius_m)
    movel([0.133874, -1.341846, -2.600787, -0.769757, 1.570796, 1.704671],accel_mss,speed_ms,0,blend_radius_m)
    movel([0.134312, -1.341959, -2.600713, -0.769717, 1.570796, 1.705108],accel_mss,speed_ms,0,blend_radius_m)
    movel([0.134537, -1.342047, -2.600656, -0.769686, 1.570796, 1.705333],accel_mss,speed_ms,0,blend_radius_m)
    movel([0.134724, -1.342134, -2.600599, -0.769656, 1.570796, 1.705520],accel_mss,speed_ms,0,blend_radius_m)
    movel([0.134889, -1.342254, -2.600521, -0.769614, 1.570796, 1.705685],accel_mss,speed_ms,0,blend_radius_m)
    movel([0.135058, -1.342462, -2.600386, -0.769541, 1.570796, 1.705854],accel_mss,speed_ms,0,blend_radius_m)
    movel([0.135120, -1.342790, -2.600172, -0.769427, 1.570796, 1.705917],accel_mss,speed_ms,0,blend_radius_m)
    movel([0.134596, -1.343303, -2.599837, -0.769249, 1.570796, 1.705392],accel_mss,speed_ms,0,blend_radius_m)
    movel([0.134152, -1.343634, -2.599621, -0.769134, 1.570796, 1.704948],accel_mss,speed_ms,0,blend_radius_m)
    movel([0.134394, -1.343806, -2.599509, -0.769074, 1.570796, 1.705190],accel_mss,speed_ms,0,blend_radius_m)
    movel([0.134638, -1.343980, -2.599395, -0.769013, 1.570796, 1.705434],accel_mss,speed_ms,0,blend_radius_m)
    movel([0.134303, -1.344283, -2.599197, -0.768908, 1.570796, 1.705100],accel_mss,speed_ms,0,blend_radius_m)
    movel([0.133995, -1.344518, -2.599044, -0.768827, 1.570796, 1.704791],accel_mss,speed_ms,0,blend_radius_m)
    movel([0.133724, -1.344655, -2.598954, -0.768780, 1.570796, 1.704520],accel_mss,speed_ms,0,blend_radius_m)
    movel([0.133806, -1.344937, -2.598770, -0.768682, 1.570796, 1.704602],accel_mss,speed_ms,0,blend_radius_m)
    movel([0.134102, -1.344945, -2.598764, -0.768679, 1.570796, 1.704899],accel_mss,speed_ms,0,blend_radius_m)
    movel([0.134405, -1.344992, -2.598733, -0.768663, 1.570796, 1.705202],accel_mss,speed_ms,0,blend_radius_m)
    movel([0.134632, -1.345146, -2.598633, -0.768610, 1.570796, 1.705428],accel_mss,speed_ms,0,blend_radius_m)
    movel([0.134781, -1.345283, -2.598543, -0.768563, 1.570796, 1.705577],accel_mss,speed_ms,0,blend_radius_m)
    movel([0.134990, -1.345391, -2.598472, -0.768526, 1.570796, 1.705786],accel_mss,speed_ms,0,blend_radius_m)
    movel([0.134941, -1.345692, -2.598275, -0.768422, 1.570796, 1.705737],accel_mss,speed_ms,0,blend_radius_m)
    movel([0.134735, -1.345909, -2.598133, -0.768347, 1.570796, 1.705532],accel_mss,speed_ms,0,blend_radius_m)
    movel([0.134593, -1.346186, -2.597951, -0.768252, 1.570796, 1.705389],accel_mss,speed_ms,0,blend_radius_m)
    movel([0.134351, -1.346477, -2.597760, -0.768152, 1.570796, 1.705148],accel_mss,speed_ms,0,blend_radius_m)
    movel([0.134008, -1.346695, -2.597616, -0.768077, 1.570796, 1.704805],accel_mss,speed_ms,0,blend_radius_m)
    movel([0.133511, -1.346849, -2.597515, -0.768024, 1.570796, 1.704307],accel_mss,speed_ms,0,blend_radius_m)
    speed_ms = 0.003
    movel([0.133372, -1.333561, -2.591198, -0.787631, 1.570796, 1.704169],accel_mss,speed_ms,0,blend_radius_m)
    speed_ms = 1.000
    movel([0.133372, -1.307920, -2.578330, -0.826139, 1.570796, 1.704169],accel_mss,speed_ms,0,blend_radius_m)
    movel([0.124146, -1.335219, -2.560894, -0.816276, 1.570796, 1.694943],accel_mss,speed_ms,0,blend_radius_m)
    movel([0.124146, -1.360403, -2.573410, -0.778576, 1.570796, 1.694943],accel_mss,speed_ms,0,blend_radius_m)
    speed_ms = 0.003
    movel([0.124146, -1.370225, -2.577968, -0.764196, 1.570796, 1.694943],accel_mss,speed_ms,0,blend_radius_m)
    speed_ms = 0.007
    movel([0.123793, -1.371087, -2.577372, -0.763930, 1.570796, 1.694589],accel_mss,speed_ms,0,blend_radius_m)
    movel([0.123280, -1.371916, -2.576797, -0.763676, 1.570796, 1.694077],accel_mss,speed_ms,0,blend_radius_m)
    movel([0.122665, -1.372875, -2.576132, -0.763382, 1.570796, 1.693461],accel_mss,speed_ms,0,blend_radius_m)
    movel([0.121838, -1.374160, -2.575237, -0.762992, 1.570796, 1.692634],accel_mss,speed_ms,0,blend_radius_m)
    movel([0.121407, -1.374875, -2.574738, -0.762775, 1.570796, 1.692203],accel_mss,speed_ms,0,blend_radius_m)
    movel([0.121174, -1.375318, -2.574429, -0.762642, 1.570796, 1.691970],accel_mss,speed_ms,0,blend_radius_m)
    movel([0.121312, -1.375503, -2.574300, -0.762586, 1.570796, 1.692108],accel_mss,speed_ms,0,blend_radius_m)
    movel([0.121589, -1.375475, -2.574320, -0.762595, 1.570796, 1.692385],accel_mss,speed_ms,0,blend_radius_m)
    movel([0.122025, -1.375385, -2.574382, -0.762621, 1.570796, 1.692821],accel_mss,speed_ms,0,blend_radius_m)
    movel([0.122716, -1.375209, -2.574505, -0.762675, 1.570796, 1.693512],accel_mss,speed_ms,0,blend_radius_m)
    movel([0.123641, -1.374975, -2.574669, -0.762745, 1.570796, 1.694437],accel_mss,speed_ms,0,blend_radius_m)
    movel([0.124044, -1.374911, -2.574713, -0.762764, 1.570796, 1.694840],accel_mss,speed_ms,0,blend_radius_m)
    movel([0.124195, -1.375102, -2.574580, -0.762707, 1.570796, 1.694992],accel_mss,speed_ms,0,blend_radius_m)
    movel([0.123079, -1.376507, -2.573598, -0.762284, 1.570796, 1.693875],accel_mss,speed_ms,0,blend_radius_m)
    movel([0.121902, -1.377963, -2.572577, -0.761849, 1.570796, 1.692699],accel_mss,speed_ms,0,blend_radius_m)
    movel([0.120523, -1.379657, -2.571385, -0.761347, 1.570796, 1.691319],accel_mss,speed_ms,0,blend_radius_m)
    movel([0.119131, -1.381360, -2.570183, -0.760846, 1.570796, 1.689928],accel_mss,speed_ms,0,blend_radius_m)
    movel([0.117908, -1.382848, -2.569129, -0.760412, 1.570796, 1.688704],accel_mss,speed_ms,0,blend_radius_m)
    movel([0.116864, -1.384114, -2.568230, -0.760045, 1.570796, 1.687661],accel_mss,speed_ms,0,blend_radius_m)
    movel([0.116633, -1.384373, -2.568045, -0.759971, 1.570796, 1.687429],accel_mss,speed_ms,0,blend_radius_m)
    movel([0.116427, -1.384584, -2.567895, -0.759910, 1.570796, 1.687224],accel_mss,speed_ms,0,blend_radius_m)
    movel([0.116381, -1.384342, -2.568068, -0.759980, 1.570796, 1.687177],accel_mss,speed_ms,0,blend_radius_m)
    movel([0.116785, -1.383473, -2.568685, -0.760231, 1.570796, 1.687582],accel_mss,speed_ms,0,blend_radius_m)
    movel([0.117268, -1.382455, -2.569408, -0.760527, 1.570796, 1.688064],accel_mss,speed_ms,0,blend_radius_m)
    movel([0.117834, -1.381287, -2.570234, -0.760868, 1.570796, 1.688631],accel_mss,speed_ms,0,blend_radius_m)
    movel([0.118529, -1.379857, -2.571244, -0.761288, 1.570796, 1.689326],accel_mss,speed_ms,0,blend_radius_m)
    movel([0.118953, -1.378940, -2.571890, -0.761559, 1.570796, 1.689749],accel_mss,speed_ms,0,blend_radius_m)
    movel([0.119224, -1.378300, -2.572340, -0.761749, 1.570796, 1.690020],accel_mss,speed_ms,0,blend_radius_m)
    movel([0.119087, -1.378136, -2.572455, -0.761798, 1.570796, 1.689884],accel_mss,speed_ms,0,blend_radius_m)
    movel([0.118747, -1.378188, -2.572418, -0.761782, 1.570796, 1.689544],accel_mss,speed_ms,0,blend_radius_m)
    movel([0.118246, -1.378296, -2.572343, -0.761750, 1.570796, 1.689042],accel_mss,speed_ms,0,blend_radius_m)
    movel([0.117501, -1.378488, -2.572208, -0.761693, 1.570796, 1.688298],accel_mss,speed_ms,0,blend_radius_m)
    movel([0.116757, -1.378680, -2.572073, -0.761636, 1.570796, 1.687553],accel_mss,speed_ms,0,blend_radius_m)
    movel([0.116258, -1.378787, -2.571997, -0.761604, 1.570796, 1.687054],accel_mss,speed_ms,0,blend_radius_m)
    movel([0.115918, -1.378840, -2.571960, -0.761589, 1.570796, 1.686714],accel_mss,speed_ms,0,blend_radius_m)
    movel([0.115788, -1.378677, -2.572075, -0.761637, 1.570796, 1.686584],accel_mss,speed_ms,0,blend_radius_m)
    movel([0.116123, -1.377916, -2.572609, -0.761863, 1.570796, 1.686920],accel_mss,speed_ms,0,blend_radius_m)
    movel([0.116612, -1.376865, -2.573347, -0.762177, 1.570796, 1.687408],accel_mss,speed_ms,0,blend_radius_m)
    movel([0.117386, -1.375283, -2.574453, -0.762652, 1.570796, 1.688182],accel_mss,speed_ms,0,blend_radius_m)
    movel([0.118051, -1.373950, -2.575383, -0.763055, 1.570796, 1.688847],accel_mss,speed_ms,0,blend_radius_m)
    movel([0.118642, -1.372791, -2.576190, -0.763408, 1.570796, 1.689439],accel_mss,speed_ms,0,blend_radius_m)
    movel([0.119160, -1.371793, -2.576883, -0.763713, 1.570796, 1.689956],accel_mss,speed_ms,0,blend_radius_m)
    movel([0.119467, -1.371483, -2.577098, -0.763808, 1.570796, 1.690263],accel_mss,speed_ms,0,blend_radius_m)
    movel([0.119865, -1.371330, -2.577204, -0.763855, 1.570796, 1.690661],accel_mss,speed_ms,0,blend_radius_m)
    movel([0.120531, -1.371128, -2.577343, -0.763917, 1.570796, 1.691328],accel_mss,speed_ms,0,blend_radius_m)
    movel([0.121831, -1.370775, -2.577588, -0.764026, 1.570796, 1.692628],accel_mss,speed_ms,0,blend_radius_m)
    movel([0.122994, -1.370473, -2.577797, -0.764119, 1.570796, 1.693790],accel_mss,speed_ms,0,blend_radius_m)
    movel([0.123692, -1.370311, -2.577909, -0.764169, 1.570796, 1.694488],accel_mss,speed_ms,0,blend_radius_m)
    movel([0.124146, -1.370225, -2.577968, -0.764196, 1.570796, 1.694943],accel_mss,speed_ms,0,blend_radius_m)
    speed_ms = 0.003
    movel([0.124146, -1.373545, -2.579471, -0.759372, 1.570796, 1.694943],accel_mss,speed_ms,0,blend_radius_m)
    speed_ms = 0.007
    movel([0.123793, -1.374405, -2.578873, -0.759111, 1.570796, 1.694589],accel_mss,speed_ms,0,blend_radius_m)
    movel([0.123280, -1.375232, -2.578297, -0.758860, 1.570796, 1.694077],accel_mss,speed_ms,0,blend_radius_m)
    movel([0.122665, -1.376188, -2.577630, -0.758571, 1.570796, 1.693461],accel_mss,speed_ms,0,blend_radius_m)
    movel([0.121838, -1.377470, -2.576733, -0.758186, 1.570796, 1.692634],accel_mss,speed_ms,0,blend_radius_m)
    movel([0.121407, -1.378183, -2.576233, -0.757972, 1.570796, 1.692203],accel_mss,speed_ms,0,blend_radius_m)
    movel([0.121174, -1.378625, -2.575924, -0.757841, 1.570796, 1.691970],accel_mss,speed_ms,0,blend_radius_m)
    movel([0.121312, -1.378810, -2.575794, -0.757786, 1.570796, 1.692108],accel_mss,speed_ms,0,blend_radius_m)
    movel([0.121589, -1.378781, -2.575814, -0.757794, 1.570796, 1.692385],accel_mss,speed_ms,0,blend_radius_m)
    movel([0.122025, -1.378692, -2.575877, -0.757821, 1.570796, 1.692821],accel_mss,speed_ms,0,blend_radius_m)
    movel([0.122716, -1.378516, -2.576000, -0.757873, 1.570796, 1.693512],accel_mss,speed_ms,0,blend_radius_m)
    movel([0.123641, -1.378282, -2.576164, -0.757943, 1.570796, 1.694437],accel_mss,speed_ms,0,blend_radius_m)
    movel([0.124044, -1.378219, -2.576208, -0.757962, 1.570796, 1.694840],accel_mss,speed_ms,0,blend_radius_m)
    movel([0.124195, -1.378409, -2.576075, -0.757905, 1.570796, 1.694992],accel_mss,speed_ms,0,blend_radius_m)
    movel([0.123079, -1.379810, -2.575090, -0.757489, 1.570796, 1.693875],accel_mss,speed_ms,0,blend_radius_m)
    movel([0.121902, -1.381262, -2.574067, -0.757060, 1.570796, 1.692699],accel_mss,speed_ms,0,blend_radius_m)
    movel([0.120523, -1.382952, -2.572872, -0.756565, 1.570796, 1.691319],accel_mss,speed_ms,0,blend_radius_m)
    movel([0.119131, -1.384650, -2.571667, -0.756072, 1.570796, 1.689928],accel_mss,speed_ms,0,blend_radius_m)
    movel([0.117908, -1.386135, -2.570610, -0.755644, 1.570796, 1.688704],accel_mss,speed_ms,0,blend_radius_m)
    movel([0.116864, -1.387397, -2.569710, -0.755283, 1.570796, 1.687661],accel_mss,speed_ms,0,blend_radius_m)
    movel([0.116633, -1.387655, -2.569525, -0.755209, 1.570796, 1.687429],accel_mss,speed_ms,0,blend_radius_m)
    movel([0.116427, -1.387865, -2.569374, -0.755149, 1.570796, 1.687224],accel_mss,speed_ms,0,blend_radius_m)
    movel([0.116381, -1.387624, -2.569547, -0.755218, 1.570796, 1.687177],accel_mss,speed_ms,0,blend_radius_m)
    movel([0.116785, -1.386757, -2.570166, -0.755465, 1.570796, 1.687582],accel_mss,speed_ms,0,blend_radius_m)
    movel([0.117268, -1.385742, -2.570890, -0.755757, 1.570796, 1.688064],accel_mss,speed_ms,0,blend_radius_m)
    movel([0.117834, -1.384578, -2.571719, -0.756093, 1.570796, 1.688631],accel_mss,speed_ms,0,blend_radius_m)
    movel([0.118529, -1.383151, -2.572731, -0.756507, 1.570796, 1.689326],accel_mss,speed_ms,0,blend_radius_m)
    movel([0.118953, -1.382237, -2.573378, -0.756774, 1.570796, 1.689749],accel_mss,speed_ms,0,blend_radius_m)
    movel([0.119224, -1.381599, -2.573829, -0.756961, 1.570796, 1.690020],accel_mss,speed_ms,0,blend_radius_m)
    movel([0.119087, -1.381435, -2.573945, -0.757009, 1.570796, 1.689884],accel_mss,speed_ms,0,blend_radius_m)
    movel([0.118747, -1.381487, -2.573908, -0.756994, 1.570796, 1.689544],accel_mss,speed_ms,0,blend_radius_m)
    movel([0.118246, -1.381595, -2.573832, -0.756962, 1.570796, 1.689042],accel_mss,speed_ms,0,blend_radius_m)
    movel([0.117501, -1.381786, -2.573697, -0.756906, 1.570796, 1.688298],accel_mss,speed_ms,0,blend_radius_m)
    movel([0.116757, -1.381977, -2.573562, -0.756850, 1.570796, 1.687553],accel_mss,speed_ms,0,blend_radius_m)
    movel([0.116258, -1.382085, -2.573486, -0.756818, 1.570796, 1.687054],accel_mss,speed_ms,0,blend_radius_m)
    movel([0.115918, -1.382138, -2.573448, -0.756803, 1.570796, 1.686714],accel_mss,speed_ms,0,blend_radius_m)
    movel([0.115788, -1.381975, -2.573563, -0.756851, 1.570796, 1.686584],accel_mss,speed_ms,0,blend_radius_m)
    movel([0.116123, -1.381216, -2.574099, -0.757073, 1.570796, 1.686920],accel_mss,speed_ms,0,blend_radius_m)
    movel([0.116612, -1.380167, -2.574839, -0.757383, 1.570796, 1.687408],accel_mss,speed_ms,0,blend_radius_m)
    movel([0.117386, -1.378590, -2.575948, -0.757851, 1.570796, 1.688182],accel_mss,speed_ms,0,blend_radius_m)
    movel([0.118051, -1.377261, -2.576880, -0.758248, 1.570796, 1.688847],accel_mss,speed_ms,0,blend_radius_m)
    movel([0.118642, -1.376105, -2.577688, -0.758596, 1.570796, 1.689439],accel_mss,speed_ms,0,blend_radius_m)
    movel([0.119160, -1.375109, -2.578383, -0.758897, 1.570796, 1.689956],accel_mss,speed_ms,0,blend_radius_m)
    movel([0.119467, -1.374800, -2.578598, -0.758991, 1.570796, 1.690263],accel_mss,speed_ms,0,blend_radius_m)
    movel([0.119865, -1.374647, -2.578705, -0.759037, 1.570796, 1.690661],accel_mss,speed_ms,0,blend_radius_m)
    movel([0.120531, -1.374446, -2.578845, -0.759098, 1.570796, 1.691328],accel_mss,speed_ms,0,blend_radius_m)
    movel([0.121831, -1.374094, -2.579090, -0.759205, 1.570796, 1.692628],accel_mss,speed_ms,0,blend_radius_m)
    movel([0.122994, -1.373793, -2.579299, -0.759297, 1.570796, 1.693790],accel_mss,speed_ms,0,blend_radius_m)
    movel([0.123692, -1.373631, -2.579411, -0.759346, 1.570796, 1.694488],accel_mss,speed_ms,0,blend_radius_m)
    movel([0.124146, -1.373545, -2.579471, -0.759372, 1.570796, 1.694943],accel_mss,speed_ms,0,blend_radius_m)
    speed_ms = 0.003
    movel([0.124146, -1.360403, -2.573410, -0.778576, 1.570796, 1.694943],accel_mss,speed_ms,0,blend_radius_m)
    speed_ms = 1.000
    movel([0.124146, -1.335219, -2.560894, -0.816276, 1.570796, 1.694943],accel_mss,speed_ms,0,blend_radius_m)
    movel([0.115988, -1.357886, -2.545671, -0.808832, 1.570796, 1.686785],accel_mss,speed_ms,0,blend_radius_m)
    movel([0.115988, -1.382667, -2.557897, -0.771824, 1.570796, 1.686785],accel_mss,speed_ms,0,blend_radius_m)
    speed_ms = 0.003
    movel([0.115988, -1.392317, -2.562347, -0.757725, 1.570796, 1.686785],accel_mss,speed_ms,0,blend_radius_m)
    speed_ms = 0.007
    movel([0.116395, -1.392329, -2.562339, -0.757721, 1.570796, 1.687191],accel_mss,speed_ms,0,blend_radius_m)
    movel([0.116711, -1.392556, -2.562174, -0.757658, 1.570796, 1.687507],accel_mss,speed_ms,0,blend_radius_m)
    movel([0.116919, -1.392985, -2.561864, -0.757540, 1.570796, 1.687715],accel_mss,speed_ms,0,blend_radius_m)
    movel([0.116976, -1.393318, -2.561623, -0.757448, 1.570796, 1.687772],accel_mss,speed_ms,0,blend_radius_m)
    movel([0.116649, -1.393630, -2.561397, -0.757362, 1.570796, 1.687445],accel_mss,speed_ms,0,blend_radius_m)
    movel([0.116200, -1.393658, -2.561377, -0.757355, 1.570796, 1.686996],accel_mss,speed_ms,0,blend_radius_m)
    movel([0.115692, -1.393625, -2.561401, -0.757364, 1.570796, 1.686488],accel_mss,speed_ms,0,blend_radius_m)
    movel([0.115348, -1.393521, -2.561476, -0.757392, 1.570796, 1.686144],accel_mss,speed_ms,0,blend_radius_m)
    movel([0.115151, -1.393344, -2.561604, -0.757441, 1.570796, 1.685947],accel_mss,speed_ms,0,blend_radius_m)
    movel([0.115085, -1.393091, -2.561788, -0.757511, 1.570796, 1.685881],accel_mss,speed_ms,0,blend_radius_m)
    movel([0.115165, -1.392773, -2.562018, -0.757598, 1.570796, 1.685962],accel_mss,speed_ms,0,blend_radius_m)
    movel([0.115516, -1.392508, -2.562209, -0.757672, 1.570796, 1.686313],accel_mss,speed_ms,0,blend_radius_m)
    movel([0.115988, -1.392317, -2.562347, -0.757725, 1.570796, 1.686785],accel_mss,speed_ms,0,blend_radius_m)
    speed_ms = 0.003
    movel([0.115988, -1.395577, -2.563814, -0.752998, 1.570796, 1.686785],accel_mss,speed_ms,0,blend_radius_m)
    speed_ms = 0.007
    movel([0.116395, -1.395589, -2.563805, -0.752995, 1.570796, 1.687191],accel_mss,speed_ms,0,blend_radius_m)
    movel([0.116711, -1.395816, -2.563641, -0.752933, 1.570796, 1.687507],accel_mss,speed_ms,0,blend_radius_m)
    movel([0.116919, -1.396243, -2.563330, -0.752816, 1.570796, 1.687715],accel_mss,speed_ms,0,blend_radius_m)
    movel([0.116976, -1.396576, -2.563088, -0.752726, 1.570796, 1.687772],accel_mss,speed_ms,0,blend_radius_m)
    movel([0.116649, -1.396886, -2.562861, -0.752641, 1.570796, 1.687445],accel_mss,speed_ms,0,blend_radius_m)
    movel([0.116200, -1.396914, -2.562841, -0.752634, 1.570796, 1.686996],accel_mss,speed_ms,0,blend_radius_m)
    movel([0.115692, -1.396881, -2.562865, -0.752643, 1.570796, 1.686488],accel_mss,speed_ms,0,blend_radius_m)
    movel([0.115348, -1.396778, -2.562940, -0.752671, 1.570796, 1.686144],accel_mss,speed_ms,0,blend_radius_m)
    movel([0.115151, -1.396601, -2.563069, -0.752719, 1.570796, 1.685947],accel_mss,speed_ms,0,blend_radius_m)
    movel([0.115085, -1.396349, -2.563253, -0.752787, 1.570796, 1.685881],accel_mss,speed_ms,0,blend_radius_m)
    movel([0.115165, -1.396032, -2.563483, -0.752874, 1.570796, 1.685962],accel_mss,speed_ms,0,blend_radius_m)
    movel([0.115516, -1.395768, -2.563675, -0.752946, 1.570796, 1.686313],accel_mss,speed_ms,0,blend_radius_m)
    movel([0.115988, -1.395577, -2.563814, -0.752998, 1.570796, 1.686785],accel_mss,speed_ms,0,blend_radius_m)
    speed_ms = 0.003
    movel([0.115988, -1.382667, -2.557897, -0.771824, 1.570796, 1.686785],accel_mss,speed_ms,0,blend_radius_m)
    speed_ms = 1.000
    movel([0.115988, -1.357886, -2.545671, -0.808832, 1.570796, 1.686785],accel_mss,speed_ms,0,blend_radius_m)
    movel([0.119782, -1.357452, -2.545969, -0.808968, 1.570796, 1.690578],accel_mss,speed_ms,0,blend_radius_m)
    movel([0.119782, -1.382241, -2.558201, -0.771947, 1.570796, 1.690578],accel_mss,speed_ms,0,blend_radius_m)
    speed_ms = 0.003
    movel([0.119782, -1.391894, -2.562653, -0.757842, 1.570796, 1.690578],accel_mss,speed_ms,0,blend_radius_m)
    speed_ms = 0.007
    movel([0.119962, -1.391564, -2.562891, -0.757933, 1.570796, 1.690759],accel_mss,speed_ms,0,blend_radius_m)
    movel([0.120193, -1.391304, -2.563079, -0.758006, 1.570796, 1.690989],accel_mss,speed_ms,0,blend_radius_m)
    movel([0.120597, -1.391186, -2.563164, -0.758039, 1.570796, 1.691393],accel_mss,speed_ms,0,blend_radius_m)
    movel([0.120783, -1.391316, -2.563070, -0.758003, 1.570796, 1.691579],accel_mss,speed_ms,0,blend_radius_m)
    movel([0.120924, -1.391495, -2.562941, -0.757953, 1.570796, 1.691720],accel_mss,speed_ms,0,blend_radius_m)
    movel([0.120906, -1.391791, -2.562728, -0.757871, 1.570796, 1.691703],accel_mss,speed_ms,0,blend_radius_m)
    movel([0.120624, -1.392181, -2.562446, -0.757762, 1.570796, 1.691420],accel_mss,speed_ms,0,blend_radius_m)
    movel([0.120435, -1.392385, -2.562298, -0.757706, 1.570796, 1.691231],accel_mss,speed_ms,0,blend_radius_m)
    movel([0.120043, -1.392729, -2.562049, -0.757611, 1.570796, 1.690839],accel_mss,speed_ms,0,blend_radius_m)
    movel([0.119669, -1.392658, -2.562101, -0.757630, 1.570796, 1.690465],accel_mss,speed_ms,0,blend_radius_m)
    movel([0.119687, -1.392232, -2.562409, -0.757748, 1.570796, 1.690484],accel_mss,speed_ms,0,blend_radius_m)
    movel([0.119782, -1.391894, -2.562653, -0.757842, 1.570796, 1.690578],accel_mss,speed_ms,0,blend_radius_m)
    speed_ms = 0.003
    movel([0.119782, -1.395155, -2.564120, -0.753113, 1.570796, 1.690578],accel_mss,speed_ms,0,blend_radius_m)
    speed_ms = 0.007
    movel([0.119962, -1.394827, -2.564359, -0.753203, 1.570796, 1.690759],accel_mss,speed_ms,0,blend_radius_m)
    movel([0.120193, -1.394568, -2.564547, -0.753275, 1.570796, 1.690989],accel_mss,speed_ms,0,blend_radius_m)
    movel([0.120597, -1.394450, -2.564632, -0.753307, 1.570796, 1.691393],accel_mss,speed_ms,0,blend_radius_m)
    movel([0.120783, -1.394579, -2.564538, -0.753271, 1.570796, 1.691579],accel_mss,speed_ms,0,blend_radius_m)
    movel([0.120924, -1.394757, -2.564409, -0.753222, 1.570796, 1.691720],accel_mss,speed_ms,0,blend_radius_m)
    movel([0.120906, -1.395052, -2.564195, -0.753141, 1.570796, 1.691703],accel_mss,speed_ms,0,blend_radius_m)
    movel([0.120624, -1.395442, -2.563912, -0.753035, 1.570796, 1.691420],accel_mss,speed_ms,0,blend_radius_m)
    movel([0.120435, -1.395645, -2.563765, -0.752979, 1.570796, 1.691231],accel_mss,speed_ms,0,blend_radius_m)
    movel([0.120043, -1.395988, -2.563515, -0.752886, 1.570796, 1.690839],accel_mss,speed_ms,0,blend_radius_m)
    movel([0.119669, -1.395917, -2.563567, -0.752905, 1.570796, 1.690465],accel_mss,speed_ms,0,blend_radius_m)
    movel([0.119687, -1.395493, -2.563875, -0.753021, 1.570796, 1.690484],accel_mss,speed_ms,0,blend_radius_m)
    movel([0.119782, -1.395155, -2.564120, -0.753113, 1.570796, 1.690578],accel_mss,speed_ms,0,blend_radius_m)
    speed_ms = 0.003
